Universal Robots PolyScope program: faichun_snake3.urp

Program faichun_snake3 (installation=default directory=/programs/snake_new createdIn=5.11.9.1010452 lastSavedIn=5.11.9.1010452 robotSerialNumber=20225200364)
Calibrated DH parameters: a=[0.00002, -0.569483, -0.54992, -0.00001, -0.000036, 0]; d=[0.180894, -146.691669, 192.918669, -46.053088, 0.119778, 0.115602]; alpha=[1.571425, -0.001534, 0.003359, 1.568739, -1.571477, 0]; deltaTheta=[0, 0.376258, -0.101074, -0.275185, -0.000002, 0]
Robot Program (runOnlyOnce=true)
  Script file /programs/FaiChun_9 Jan_11_2_t1_2.script
    | def Machining1():
    |   # Default parameters:
    |   global speed_ms = 0.05
    |   global speed_rads = 0.75
    |   global accel_mss = 3
    |   global accel_radss = 1.2
    |   global blend_radius_m = 0.0003
    | 
    |   # Add subprograms here
    |   # Start of main program
    |   # Program generated by RoboDK v5.6.8 for UR10e on 17/01/2025 17:23:54
    |   # Using nominal kinematics.
    |   blend_radius_m = 0.0003
    |   speed_ms = 0.05
    |   # set_reference(p[0.340000, -0.238000, 0.001500, 0.000000, 0.000000, 0.000000])
    |   set_tcp(p[0.000000, 0.000000, 0.252000, 0.000000, 0.000000, 0.000000])
    |   # Show Tool
    |   movej([0.145114, -1.397514, -2.446396, -0.868479, 1.570796, 1.715910],accel_radss,speed_rads,0,blend_radius_m)
    |   movel([0.145114, -1.450226, -2.476289, -0.785874, 1.570796, 1.715910],accel_mss,speed_ms,0,blend_radius_m)
    |   #SetTool1
    |   #M_RunCode6
    |   #SetRPM60000
    |   speed_ms = 0.05
    |   #M_RunCode3
    |   movel([0.145114, -1.473196, -2.487384, -0.751808, 1.570796, 1.715910],accel_mss,speed_ms,0,blend_radius_m)
    |   speed_ms = 0.003
    |   movel([0.145114, -1.479129, -2.490086, -0.743174, 1.570796, 1.715910],accel_mss,speed_ms,0,blend_radius_m)
    |   speed_ms = 0.05
    |   movel([-0.131626, -1.561533, -2.414291, -0.736565, 1.570796, 1.439170],accel_mss,speed_ms,0,blend_radius_m)
    |   movel([-0.177704, -1.331249, -2.600139, -0.781001, 1.570796, 1.393092],accel_mss,speed_ms,0,blend_radius_m)
    |   movel([0.204954, -1.166991, -2.688242, -0.857156, 1.570796, 1.775750],accel_mss,speed_ms,0,blend_radius_m)
    |   movel([0.145114, -1.479129, -2.490086, -0.743174, 1.570796, 1.715910],accel_mss,speed_ms,0,blend_radius_m)
    |   speed_ms = 0.003
    |   movel([0.145114, -1.473196, -2.487384, -0.751808, 1.570796, 1.715910],accel_mss,speed_ms,0,blend_radius_m)
    |   speed_ms = 0.05
    |   movel([0.145114, -1.450226, -2.476289, -0.785874, 1.570796, 1.715910],accel_mss,speed_ms,0,blend_radius_m)
    |   #M_RunCode9
    |   movel([0.141001, -1.443521, -2.481739, -0.787129, 1.570796, 1.711798],accel_mss,speed_ms,0,blend_radius_m)
    |   #M_RunCode3
    |   movel([0.141001, -1.466629, -2.492914, -0.752846, 1.570796, 1.711798],accel_mss,speed_ms,0,blend_radius_m)
    |   speed_ms = 0.003
    |   movel([0.141001, -1.472599, -2.495635, -0.744154, 1.570796, 1.711798],accel_mss,speed_ms,0,blend_radius_m)
    |   speed_ms = 0.012
    |   movel([0.136639, -1.473494, -2.494879, -0.744016, 1.570796, 1.707435],accel_mss,speed_ms,0,blend_radius_m)
    |   movel([0.136042, -1.477254, -2.491686, -0.743449, 1.570796, 1.706838],accel_mss,speed_ms,0,blend_radius_m)
    |   movel([0.129615, -1.478592, -2.490545, -0.743252, 1.570796, 1.700411],accel_mss,speed_ms,0,blend_radius_m)
    |   movel([0.130181, -1.474842, -2.493736, -0.743810, 1.570796, 1.700977],accel_mss,speed_ms,0,blend_radius_m)
    |   movel([0.127919, -1.475323, -2.493329, -0.743738, 1.570796, 1.698716],accel_mss,speed_ms,0,blend_radius_m)
    |   movel([0.127361, -1.479068, -2.490138, -0.743183, 1.570796, 1.698157],accel_mss,speed_ms,0,blend_radius_m)
    |   movel([0.121982, -1.480222, -2.489150, -0.743016, 1.570796, 1.692778],accel_mss,speed_ms,0,blend_radius_m)
    |   movel([0.120939, -1.480446, -2.488958, -0.742984, 1.570796, 1.691735],accel_mss,speed_ms,0,blend_radius_m)
    |   movel([0.121724, -1.474915, -2.493675, -0.743799, 1.570796, 1.692520],accel_mss,speed_ms,0,blend_radius_m)
    |   movel([0.126089, -1.473968, -2.494478, -0.743944, 1.570796, 1.696886],accel_mss,speed_ms,0,blend_radius_m)
    |   movel([0.126378, -1.472012, -2.496131, -0.744246, 1.570796, 1.697174],accel_mss,speed_ms,0,blend_radius_m)
    |   movel([0.119733, -1.473463, -2.494905, -0.744021, 1.570796, 1.690529],accel_mss,speed_ms,0,blend_radius_m)
    |   movel([0.118690, -1.480938, -2.488537, -0.742914, 1.570796, 1.689486],accel_mss,speed_ms,0,blend_radius_m)
    |   movel([0.117647, -1.481168, -2.488339, -0.742882, 1.570796, 1.688443],accel_mss,speed_ms,0,blend_radius_m)
    |   speed_ms = 0.02
    |   movel([0.002864, -1.511155, -2.461903, -0.739330, 1.570796, 1.573661],accel_mss,speed_ms,0,blend_radius_m)
    |   movel([-0.108286, -1.549104, -2.426413, -0.736872, 1.570796, 1.462510],accel_mss,speed_ms,0,blend_radius_m)
    |   speed_ms = 0.012
    |   movel([-0.109170, -1.542784, -2.432482, -0.737123, 1.570796, 1.461626],accel_mss,speed_ms,0,blend_radius_m)
    |   movel([-0.115268, -1.545135, -2.430232, -0.737022, 1.570796, 1.455529],accel_mss,speed_ms,0,blend_radius_m)
    |   movel([-0.115029, -1.546770, -2.428662, -0.736957, 1.570796, 1.455767],accel_mss,speed_ms,0,blend_radius_m)
    |   movel([-0.111023, -1.545226, -2.430145, -0.737018, 1.570796, 1.459773],accel_mss,speed_ms,0,blend_radius_m)
    |   movel([-0.110365, -1.549892, -2.425652, -0.736845, 1.570796, 1.460431],accel_mss,speed_ms,0,blend_radius_m)
    |   movel([-0.111325, -1.550258, -2.425297, -0.736833, 1.570796, 1.459472],accel_mss,speed_ms,0,blend_radius_m)
    |   movel([-0.116260, -1.552156, -2.423459, -0.736774, 1.570796, 1.454536],accel_mss,speed_ms,0,blend_radius_m)
    |   movel([-0.116726, -1.549025, -2.426489, -0.736875, 1.570796, 1.454070],accel_mss,speed_ms,0,blend_radius_m)
    |   movel([-0.118795, -1.549827, -2.425715, -0.736847, 1.570796, 1.452001],accel_mss,speed_ms,0,blend_radius_m)
    |   movel([-0.118321, -1.552953, -2.422685, -0.736751, 1.570796, 1.452475],accel_mss,speed_ms,0,blend_radius_m)
    |   movel([-0.124187, -1.555237, -2.420462, -0.736690, 1.570796, 1.446609],accel_mss,speed_ms,0,blend_radius_m)
    |   movel([-0.124683, -1.552129, -2.423485, -0.736775, 1.570796, 1.446114],accel_mss,speed_ms,0,blend_radius_m)
    |   movel([-0.128648, -1.553694, -2.421965, -0.736730, 1.570796, 1.442148],accel_mss,speed_ms,0,blend_radius_m)
    |   movel([-0.129411, -1.549091, -2.426425, -0.736873, 1.570796, 1.441385],accel_mss,speed_ms,0,blend_radius_m)
    |   movel([-0.125425, -1.547510, -2.427949, -0.736929, 1.570796, 1.445371],accel_mss,speed_ms,0,blend_radius_m)
    |   movel([-0.125687, -1.545886, -2.429511, -0.736992, 1.570796, 1.445109],accel_mss,speed_ms,0,blend_radius_m)
    |   movel([-0.129681, -1.547471, -2.427987, -0.736931, 1.570796, 1.441115],accel_mss,speed_ms,0,blend_radius_m)
    |   movel([-0.130331, -1.543596, -2.431706, -0.737087, 1.570796, 1.440465],accel_mss,speed_ms,0,blend_radius_m)
    |   movel([-0.130456, -1.542840, -2.432429, -0.737120, 1.570796, 1.440341],accel_mss,speed_ms,0,blend_radius_m)
    |   movel([-0.124505, -1.540465, -2.434693, -0.737231, 1.570796, 1.446291],accel_mss,speed_ms,0,blend_radius_m)
    |   movel([-0.124003, -1.543613, -2.431690, -0.737086, 1.570796, 1.446793],accel_mss,speed_ms,0,blend_radius_m)
    |   movel([-0.121918, -1.542790, -2.432476, -0.737122, 1.570796, 1.448878],accel_mss,speed_ms,0,blend_radius_m)
    |   movel([-0.122672, -1.537996, -2.437038, -0.737355, 1.570796, 1.448124],accel_mss,speed_ms,0,blend_radius_m)
    |   movel([-0.130730, -1.541209, -2.433985, -0.737195, 1.570796, 1.440067],accel_mss,speed_ms,0,blend_radius_m)
    |   movel([-0.146735, -1.452072, -2.512652, -0.747665, 1.570796, 1.424062],accel_mss,speed_ms,0,blend_radius_m)
    |   speed_ms = 0.02
    |   movel([-0.166789, -1.353893, -2.585329, -0.773167, 1.570796, 1.404008],accel_mss,speed_ms,0,blend_radius_m)
    |   movel([-0.166990, -1.352958, -2.585955, -0.773476, 1.570796, 1.403806],accel_mss,speed_ms,0,blend_radius_m)
    |   speed_ms = 0.012
    |   movel([-0.156896, -1.347760, -2.589410, -0.775219, 1.570796, 1.413900],accel_mss,speed_ms,0,blend_radius_m)
    |   movel([-0.158123, -1.341762, -2.593351, -0.777277, 1.570796, 1.412674],accel_mss,speed_ms,0,blend_radius_m)
    |   movel([-0.160766, -1.343128, -2.592457, -0.776804, 1.570796, 1.410031],accel_mss,speed_ms,0,blend_radius_m)
    |   movel([-0.159947, -1.347068, -2.589867, -0.775454, 1.570796, 1.410849],accel_mss,speed_ms,0,blend_radius_m)
    |   movel([-0.167424, -1.350932, -2.587305, -0.774151, 1.570796, 1.403372],accel_mss,speed_ms,0,blend_radius_m)
    |   movel([-0.167629, -1.349998, -2.587927, -0.774464, 1.570796, 1.403168],accel_mss,speed_ms,0,blend_radius_m)
    |   movel([-0.168693, -1.345153, -2.591129, -0.776107, 1.570796, 1.402103],accel_mss,speed_ms,0,blend_radius_m)
    |   movel([-0.163615, -1.342502, -2.592867, -0.777020, 1.570796, 1.407181],accel_mss,speed_ms,0,blend_radius_m)
    |   movel([-0.164053, -1.340454, -2.594203, -0.777732, 1.570796, 1.406744],accel_mss,speed_ms,0,blend_radius_m)
    |   movel([-0.169143, -1.343118, -2.592464, -0.776807, 1.570796, 1.401654],accel_mss,speed_ms,0,blend_radius_m)
    |   movel([-0.170437, -1.337285, -2.596260, -0.778844, 1.570796, 1.400359],accel_mss,speed_ms,0,blend_radius_m)
    |   movel([-0.165313, -1.334580, -2.598005, -0.779805, 1.570796, 1.405484],accel_mss,speed_ms,0,blend_radius_m)
    |   movel([-0.166173, -1.330591, -2.600559, -0.781239, 1.570796, 1.404623],accel_mss,speed_ms,0,blend_radius_m)
    |   movel([-0.158508, -1.326548, -2.603127, -0.782714, 1.570796, 1.412289],accel_mss,speed_ms,0,blend_radius_m)
    |   movel([-0.157682, -1.330578, -2.600567, -0.781243, 1.570796, 1.413114],accel_mss,speed_ms,0,blend_radius_m)
    |   movel([-0.154998, -1.329179, -2.601459, -0.781752, 1.570796, 1.415798],accel_mss,speed_ms,0,blend_radius_m)
    |   movel([-0.155811, -1.325133, -2.604020, -0.783236, 1.570796, 1.414985],accel_mss,speed_ms,0,blend_radius_m)
    |   movel([-0.148083, -1.321101, -2.606551, -0.784737, 1.570796, 1.422714],accel_mss,speed_ms,0,blend_radius_m)
    |   movel([-0.146935, -1.327148, -2.602747, -0.782494, 1.570796, 1.423861],accel_mss,speed_ms,0,blend_radius_m)
    |   movel([-0.152123, -1.329828, -2.601046, -0.781516, 1.570796, 1.418673],accel_mss,speed_ms,0,blend_radius_m)
    |   movel([-0.151712, -1.331924, -2.599708, -0.780757, 1.570796, 1.419084],accel_mss,speed_ms,0,blend_radius_m)
    |   movel([-0.143841, -1.327877, -2.602285, -0.782227, 1.570796, 1.426955],accel_mss,speed_ms,0,blend_radius_m)
    |   movel([-0.145364, -1.319691, -2.607431, -0.785267, 1.570796, 1.425432],accel_mss,speed_ms,0,blend_radius_m)
    |   movel([0.003920, -1.248574, -2.648506, -0.815310, 1.570796, 1.574716],accel_mss,speed_ms,0,blend_radius_m)
    |   speed_ms = 0.02
    |   movel([0.165154, -1.186625, -2.679348, -0.846417, 1.570796, 1.735951],accel_mss,speed_ms,0,blend_radius_m)
    |   movel([0.163152, -1.198149, -2.673935, -0.840305, 1.570796, 1.733948],accel_mss,speed_ms,0,blend_radius_m)
    |   speed_ms = 0.012
    |   movel([0.172319, -1.195184, -2.675341, -0.841863, 1.570796, 1.743115],accel_mss,speed_ms,0,blend_radius_m)
    |   movel([0.172866, -1.192193, -2.676750, -0.843445, 1.570796, 1.743662],accel_mss,speed_ms,0,blend_radius_m)
    |   movel([0.166811, -1.194153, -2.675828, -0.842408, 1.570796, 1.737608],accel_mss,speed_ms,0,blend_radius_m)
    |   movel([0.168335, -1.185580, -2.679831, -0.846978, 1.570796, 1.739131],accel_mss,speed_ms,0,blend_radius_m)
    |   movel([0.169806, -1.185096, -2.680055, -0.847238, 1.570796, 1.740602],accel_mss,speed_ms,0,blend_radius_m)
    |   movel([0.177391, -1.182622, -2.681194, -0.848573, 1.570796, 1.748187],accel_mss,speed_ms,0,blend_radius_m)
    |   movel([0.176304, -1.188464, -2.678494, -0.845432, 1.570796, 1.747100],accel_mss,speed_ms,0,blend_radius_m)
    |   movel([0.179460, -1.187457, -2.678962, -0.845971, 1.570796, 1.750256],accel_mss,speed_ms,0,blend_radius_m)
    |   movel([0.180574, -1.181595, -2.681665, -0.849129, 1.570796, 1.751371],accel_mss,speed_ms,0,blend_radius_m)
    |   movel([0.189651, -1.178707, -2.682983, -0.850699, 1.570796, 1.760447],accel_mss,speed_ms,0,blend_radius_m)
    |   movel([0.188481, -1.184611, -2.680279, -0.847499, 1.570796, 1.759277],accel_mss,speed_ms,0,blend_radius_m)
    |   movel([0.194577, -1.182720, -2.681149, -0.848520, 1.570796, 1.765374],accel_mss,speed_ms,0,blend_radius_m)
    |   movel([0.192814, -1.191401, -2.677122, -0.843866, 1.570796, 1.763610],accel_mss,speed_ms,0,blend_radius_m)
    |   movel([0.186775, -1.193250, -2.676254, -0.842885, 1.570796, 1.757572],accel_mss,speed_ms,0,blend_radius_m)
    |   movel([0.186185, -1.196251, -2.674837, -0.841302, 1.570796, 1.756982],accel_mss,speed_ms,0,blend_radius_m)
    |   movel([0.192203, -1.194418, -2.675703, -0.842268, 1.570796, 1.762999],accel_mss,speed_ms,0,blend_radius_m)
    |   movel([0.190761, -1.201563, -2.672304, -0.838522, 1.570796, 1.761557],accel_mss,speed_ms,0,blend_radius_m)
    |   movel([0.190484, -1.202941, -2.671643, -0.837806, 1.570796, 1.761280],accel_mss,speed_ms,0,blend_radius_m)
    |   movel([0.181657, -1.205609, -2.670355, -0.836426, 1.570796, 1.752453],accel_mss,speed_ms,0,blend_radius_m)
    |   movel([0.182758, -1.199906, -2.673098, -0.839385, 1.570796, 1.753554],accel_mss,speed_ms,0,blend_radius_m)
    |   movel([0.179644, -1.200868, -2.672637, -0.838884, 1.570796, 1.750441],accel_mss,speed_ms,0,blend_radius_m)
    |   movel([0.178007, -1.209492, -2.668466, -0.834430, 1.570796, 1.748803],accel_mss,speed_ms,0,blend_radius_m)
    |   movel([0.189888, -1.205903, -2.670212, -0.836273, 1.570796, 1.760685],accel_mss,speed_ms,0,blend_radius_m)
    |   speed_ms = 0.02
    |   movel([0.163402, -1.343756, -2.592046, -0.776587, 1.570796, 1.734198],accel_mss,speed_ms,0,blend_radius_m)
    |   movel([0.143535, -1.457310, -2.508372, -0.746708, 1.570796, 1.714331],accel_mss,speed_ms,0,blend_radius_m)
    |   speed_ms = 0.012
    |   movel([0.134639, -1.459191, -2.506824, -0.746374, 1.570796, 1.705436],accel_mss,speed_ms,0,blend_radius_m)
    |   movel([0.133732, -1.465007, -2.502005, -0.745377, 1.570796, 1.704528],accel_mss,speed_ms,0,blend_radius_m)
    |   movel([0.136023, -1.464522, -2.502409, -0.745459, 1.570796, 1.706819],accel_mss,speed_ms,0,blend_radius_m)
    |   movel([0.136629, -1.460695, -2.505582, -0.746111, 1.570796, 1.707425],accel_mss,speed_ms,0,blend_radius_m)
    |   movel([0.143192, -1.459319, -2.506719, -0.746352, 1.570796, 1.713988],accel_mss,speed_ms,0,blend_radius_m)
    |   movel([0.143038, -1.460245, -2.505954, -0.746190, 1.570796, 1.713835],accel_mss,speed_ms,0,blend_radius_m)
    |   movel([0.142251, -1.464999, -2.502011, -0.745379, 1.570796, 1.713048],accel_mss,speed_ms,0,blend_radius_m)
    |   movel([0.137849, -1.465911, -2.501251, -0.745227, 1.570796, 1.708646],accel_mss,speed_ms,0,blend_radius_m)
    |   movel([0.137533, -1.467886, -2.499600, -0.744903, 1.570796, 1.708330],accel_mss,speed_ms,0,blend_radius_m)
    |   movel([0.141927, -1.466979, -2.500359, -0.745051, 1.570796, 1.712723],accel_mss,speed_ms,0,blend_radius_m)
    |   movel([0.141001, -1.472599, -2.495635, -0.744154, 1.570796, 1.711798],accel_mss,speed_ms,0,blend_radius_m)
    |   speed_ms = 0.003
    |   movel([0.141001, -1.466629, -2.492914, -0.752846, 1.570796, 1.711798],accel_mss,speed_ms,0,blend_radius_m)
    |   speed_ms = 0.05
    |   movel([0.141001, -1.443521, -2.481739, -0.787129, 1.570796, 1.711798],accel_mss,speed_ms,0,blend_radius_m)
    |   #M_RunCode9
    |   movel([-0.095971, -1.320143, -2.570643, -0.821603, 1.570796, 1.474826],accel_mss,speed_ms,0,blend_radius_m)
    |   #M_RunCode3
    |   # num 0 inside
    |   movel([-0.095971, -1.345583, -2.583353, -0.783454, 1.570796, 1.474826],accel_mss,speed_ms,0,blend_radius_m)
    |   speed_ms = 0.003
    |   movel([-0.095971, -1.352203, -2.586459, -0.773727, 1.570796, 1.474826],accel_mss,speed_ms,0,blend_radius_m)
    |   speed_ms = 0.015
    |   movel([-0.101060, -1.358991, -2.581897, -0.771501, 1.570796, 1.469736],accel_mss,speed_ms,0,blend_radius_m)
    |   movel([-0.105019, -1.363609, -2.578758, -0.770023, 1.570796, 1.465778],accel_mss,speed_ms,0,blend_radius_m)
    |   movel([-0.106639, -1.365123, -2.577722, -0.769544, 1.570796, 1.464157],accel_mss,speed_ms,0,blend_radius_m)
    |   movel([-0.108096, -1.366111, -2.577044, -0.769234, 1.570796, 1.462701],accel_mss,speed_ms,0,blend_radius_m)
    |   movel([-0.109388, -1.366578, -2.576723, -0.769088, 1.570796, 1.461409],accel_mss,speed_ms,0,blend_radius_m)
    |   movel([-0.110520, -1.366524, -2.576760, -0.769105, 1.570796, 1.460276],accel_mss,speed_ms,0,blend_radius_m)
    |   movel([-0.111321, -1.366002, -2.577119, -0.769268, 1.570796, 1.459475],accel_mss,speed_ms,0,blend_radius_m)
    |   movel([-0.111616, -1.365061, -2.577764, -0.769564, 1.570796, 1.459180],accel_mss,speed_ms,0,blend_radius_m)
    |   movel([-0.111403, -1.363700, -2.578696, -0.769994, 1.570796, 1.459393],accel_mss,speed_ms,0,blend_radius_m)
    |   movel([-0.110683, -1.361913, -2.579914, -0.770562, 1.570796, 1.460113],accel_mss,speed_ms,0,blend_radius_m)
    |   movel([-0.107823, -1.356944, -2.583280, -0.772165, 1.570796, 1.462973],accel_mss,speed_ms,0,blend_radius_m)
    |   movel([-0.103126, -1.350010, -2.587919, -0.774460, 1.570796, 1.467671],accel_mss,speed_ms,0,blend_radius_m)
    |   movel([-0.097993, -1.343109, -2.592470, -0.776810, 1.570796, 1.472803],accel_mss,speed_ms,0,blend_radius_m)
    |   movel([-0.093909, -1.338331, -2.595583, -0.778476, 1.570796, 1.476888],accel_mss,speed_ms,0,blend_radius_m)
    |   movel([-0.092221, -1.336752, -2.596604, -0.779033, 1.570796, 1.478576],accel_mss,speed_ms,0,blend_radius_m)
    |   movel([-0.090706, -1.335718, -2.597272, -0.779399, 1.570796, 1.480090],accel_mss,speed_ms,0,blend_radius_m)
    |   movel([-0.089366, -1.335233, -2.597584, -0.779572, 1.570796, 1.481430],accel_mss,speed_ms,0,blend_radius_m)
    |   movel([-0.088203, -1.335298, -2.597543, -0.779549, 1.570796, 1.482593],accel_mss,speed_ms,0,blend_radius_m)
    |   movel([-0.087396, -1.335857, -2.597182, -0.779350, 1.570796, 1.483400],accel_mss,speed_ms,0,blend_radius_m)
    |   movel([-0.087120, -1.336850, -2.596541, -0.778998, 1.570796, 1.483676],accel_mss,speed_ms,0,blend_radius_m)
    |   movel([-0.087378, -1.338279, -2.595616, -0.778494, 1.570796, 1.483418],accel_mss,speed_ms,0,blend_radius_m)
    |   movel([-0.088162, -1.340134, -2.594412, -0.777843, 1.570796, 1.482634],accel_mss,speed_ms,0,blend_radius_m)
    |   movel([-0.091172, -1.345231, -2.591077, -0.776081, 1.570796, 1.479624],accel_mss,speed_ms,0,blend_radius_m)
    |   movel([-0.095971, -1.352203, -2.586459, -0.773727, 1.570796, 1.474826],accel_mss,speed_ms,0,blend_radius_m)
    |   speed_ms = 0.003
    |   movel([-0.095971, -1.345583, -2.583353, -0.783454, 1.570796, 1.474826],accel_mss,speed_ms,0,blend_radius_m)
    |   speed_ms = 0.05
    |   movel([-0.095971, -1.320143, -2.570643, -0.821603, 1.570796, 1.474826],accel_mss,speed_ms,0,blend_radius_m)
    |   #M_RunCode9
    |   movel([-0.088305, -1.322635, -2.569052, -0.820702, 1.570796, 1.482491],accel_mss,speed_ms,0,blend_radius_m)
    |   #M_RunCode3
    |   #num 0 outside
    |   movel([-0.088305, -1.348033, -2.581729, -0.782626, 1.570796, 1.482491],accel_mss,speed_ms,0,blend_radius_m)
    |   speed_ms = 0.003
    |   movel([-0.088305, -1.354642, -2.584827, -0.772920, 1.570796, 1.482491],accel_mss,speed_ms,0,blend_radius_m)
    |   speed_ms = 0.015
    |   movel([-0.090204, -1.357095, -2.583178, -0.772116, 1.570796, 1.480592],accel_mss,speed_ms,0,blend_radius_m)
    |   movel([-0.092146, -1.359299, -2.581689, -0.771401, 1.570796, 1.478650],accel_mss,speed_ms,0,blend_radius_m)
    |   movel([-0.094134, -1.361259, -2.580359, -0.770771, 1.570796, 1.476662],accel_mss,speed_ms,0,blend_radius_m)
    |   movel([-0.096168, -1.362974, -2.579191, -0.770224, 1.570796, 1.474629],accel_mss,speed_ms,0,blend_radius_m)
    |   movel([-0.098207, -1.364435, -2.578193, -0.769761, 1.570796, 1.472589],accel_mss,speed_ms,0,blend_radius_m)
    |   movel([-0.100213, -1.365632, -2.577372, -0.769384, 1.570796, 1.470584],accel_mss,speed_ms,0,blend_radius_m)
    |   movel([-0.102186, -1.366569, -2.576729, -0.769091, 1.570796, 1.468610],accel_mss,speed_ms,0,blend_radius_m)
    |   movel([-0.104128, -1.367242, -2.576266, -0.768881, 1.570796, 1.466669],accel_mss,speed_ms,0,blend_radius_m)
    |   movel([-0.106011, -1.367658, -2.575980, -0.768751, 1.570796, 1.464785],accel_mss,speed_ms,0,blend_radius_m)
    |   movel([-0.107803, -1.367820, -2.575868, -0.768701, 1.570796, 1.462993],accel_mss,speed_ms,0,blend_radius_m)
    |   movel([-0.109510, -1.367730, -2.575930, -0.768729, 1.570796, 1.461286],accel_mss,speed_ms,0,blend_radius_m)
    |   movel([-0.111131, -1.367388, -2.576166, -0.768835, 1.570796, 1.459665],accel_mss,speed_ms,0,blend_radius_m)
    |   movel([-0.112591, -1.366814, -2.576561, -0.769014, 1.570796, 1.458205],accel_mss,speed_ms,0,blend_radius_m)
    |   movel([-0.113810, -1.366033, -2.577098, -0.769259, 1.570796, 1.456987],accel_mss,speed_ms,0,blend_radius_m)
    |   movel([-0.114791, -1.365044, -2.577776, -0.769569, 1.570796, 1.456006],accel_mss,speed_ms,0,blend_radius_m)
    |   movel([-0.115530, -1.363841, -2.578599, -0.769949, 1.570796, 1.455266],accel_mss,speed_ms,0,blend_radius_m)
    |   movel([-0.116005, -1.362439, -2.579556, -0.770394, 1.570796, 1.454792],accel_mss,speed_ms,0,blend_radius_m)
    |   movel([-0.116190, -1.360849, -2.580638, -0.770902, 1.570796, 1.454606],accel_mss,speed_ms,0,blend_radius_m)
    |   movel([-0.116085, -1.359067, -2.581846, -0.771476, 1.570796, 1.454711],accel_mss,speed_ms,0,blend_radius_m)
    |   movel([-0.115685, -1.357091, -2.583180, -0.772117, 1.570796, 1.455111],accel_mss,speed_ms,0,blend_radius_m)
    |   movel([-0.114980, -1.354950, -2.584621, -0.772819, 1.570796, 1.455816],accel_mss,speed_ms,0,blend_radius_m)
    |   movel([-0.113953, -1.352671, -2.586146, -0.773572, 1.570796, 1.456843],accel_mss,speed_ms,0,blend_radius_m)
    |   movel([-0.112603, -1.350256, -2.587755, -0.774378, 1.570796, 1.458193],accel_mss,speed_ms,0,blend_radius_m)
    |   movel([-0.110928, -1.347704, -2.589447, -0.775238, 1.570796, 1.459868],accel_mss,speed_ms,0,blend_radius_m)
    |   movel([-0.109051, -1.345192, -2.591103, -0.776094, 1.570796, 1.461745],accel_mss,speed_ms,0,blend_radius_m)
    |   movel([-0.107107, -1.342916, -2.592596, -0.776877, 1.570796, 1.463689],accel_mss,speed_ms,0,blend_radius_m)
    |   movel([-0.105094, -1.340873, -2.593931, -0.777586, 1.570796, 1.465702],accel_mss,speed_ms,0,blend_radius_m)
    |   movel([-0.103017, -1.339070, -2.595103, -0.778216, 1.570796, 1.467780],accel_mss,speed_ms,0,blend_radius_m)
    |   movel([-0.100919, -1.337525, -2.596105, -0.778759, 1.570796, 1.469878],accel_mss,speed_ms,0,blend_radius_m)
    |   movel([-0.098849, -1.336258, -2.596923, -0.779208, 1.570796, 1.471947],accel_mss,speed_ms,0,blend_radius_m)
    |   movel([-0.096809, -1.335267, -2.597562, -0.779560, 1.570796, 1.473987],accel_mss,speed_ms,0,blend_radius_m)
    |   movel([-0.094800, -1.334558, -2.598018, -0.779812, 1.570796, 1.475997],accel_mss,speed_ms,0,blend_radius_m)
    |   movel([-0.092856, -1.334126, -2.598296, -0.779966, 1.570796, 1.477940],accel_mss,speed_ms,0,blend_radius_m)
    |   movel([-0.091005, -1.333963, -2.598401, -0.780025, 1.570796, 1.479791],accel_mss,speed_ms,0,blend_radius_m)
    |   movel([-0.089247, -1.334068, -2.598334, -0.779987, 1.570796, 1.481550],accel_mss,speed_ms,0,blend_radius_m)
    |   movel([-0.087589, -1.334445, -2.598091, -0.779853, 1.570796, 1.483208],accel_mss,speed_ms,0,blend_radius_m)
    |   movel([-0.086106, -1.335067, -2.597691, -0.779631, 1.570796, 1.484690],accel_mss,speed_ms,0,blend_radius_m)
    |   movel([-0.084880, -1.335904, -2.597152, -0.779333, 1.570796, 1.485916],accel_mss,speed_ms,0,blend_radius_m)
    |   movel([-0.083910, -1.336959, -2.596471, -0.778959, 1.570796, 1.486886],accel_mss,speed_ms,0,blend_radius_m)
    |   movel([-0.083195, -1.338228, -2.595649, -0.778512, 1.570796, 1.487601],accel_mss,speed_ms,0,blend_radius_m)
    |   movel([-0.082761, -1.339697, -2.594696, -0.777996, 1.570796, 1.488035],accel_mss,speed_ms,0,blend_radius_m)
    |   movel([-0.082632, -1.341356, -2.593615, -0.777417, 1.570796, 1.488165],accel_mss,speed_ms,0,blend_radius_m)
    |   movel([-0.082808, -1.343205, -2.592407, -0.776777, 1.570796, 1.487989],accel_mss,speed_ms,0,blend_radius_m)
    |   movel([-0.083285, -1.345236, -2.591074, -0.776079, 1.570796, 1.487512],accel_mss,speed_ms,0,blend_radius_m)
    |   movel([-0.084070, -1.347416, -2.589637, -0.775336, 1.570796, 1.486727],accel_mss,speed_ms,0,blend_radius_m)
    |   movel([-0.085171, -1.349713, -2.588116, -0.774560, 1.570796, 1.485626],accel_mss,speed_ms,0,blend_radius_m)
    |   movel([-0.086583, -1.352122, -2.586513, -0.773754, 1.570796, 1.484213],accel_mss,speed_ms,0,blend_radius_m)
    |   movel([-0.088305, -1.354642, -2.584827, -0.772920, 1.570796, 1.482491],accel_mss,speed_ms,0,blend_radius_m)
    |   speed_ms = 0.003
    |   movel([-0.088305, -1.348033, -2.581729, -0.782626, 1.570796, 1.482491],accel_mss,speed_ms,0,blend_radius_m)
    |   speed_ms = 0.05
    |   movel([-0.088305, -1.322635, -2.569052, -0.820702, 1.570796, 1.482491],accel_mss,speed_ms,0,blend_radius_m)
    |   #M_RunCode9
    |   movel([-0.118832, -1.321958, -2.569485, -0.820946, 1.570796, 1.451964],accel_mss,speed_ms,0,blend_radius_m)
    |   #M_RunCode3
    |   movel([-0.118832, -1.347368, -2.582171, -0.782850, 1.570796, 1.451964],accel_mss,speed_ms,0,blend_radius_m)
    |   speed_ms = 0.003
    |   movel([-0.118832, -1.353979, -2.585271, -0.773138, 1.570796, 1.451964],accel_mss,speed_ms,0,blend_radius_m)
    |   speed_ms = 0.02
    |   movel([-0.124934, -1.362775, -2.579327, -0.770287, 1.570796, 1.445862],accel_mss,speed_ms,0,blend_radius_m)
    |   movel([-0.148632, -1.356620, -2.583498, -0.772271, 1.570796, 1.422164],accel_mss,speed_ms,0,blend_radius_m)
    |   movel([-0.148043, -1.355734, -2.584094, -0.772561, 1.570796, 1.422754],accel_mss,speed_ms,0,blend_radius_m)
    |   movel([-0.146262, -1.353538, -2.585567, -0.773284, 1.570796, 1.424534],accel_mss,speed_ms,0,blend_radius_m)
    |   movel([-0.143953, -1.351516, -2.586917, -0.773956, 1.570796, 1.426844],accel_mss,speed_ms,0,blend_radius_m)
    |   movel([-0.141315, -1.349690, -2.588131, -0.774568, 1.570796, 1.429481],accel_mss,speed_ms,0,blend_radius_m)
    |   movel([-0.138559, -1.348086, -2.589194, -0.775109, 1.570796, 1.432238],accel_mss,speed_ms,0,blend_radius_m)
    |   movel([-0.130967, -1.344319, -2.591676, -0.776393, 1.570796, 1.439829],accel_mss,speed_ms,0,blend_radius_m)
    |   movel([-0.123880, -1.340890, -2.593919, -0.777580, 1.570796, 1.446916],accel_mss,speed_ms,0,blend_radius_m)
    |   movel([-0.121261, -1.339412, -2.594881, -0.778096, 1.570796, 1.449535],accel_mss,speed_ms,0,blend_radius_m)
    |   movel([-0.118795, -1.337754, -2.595956, -0.778678, 1.570796, 1.452001],accel_mss,speed_ms,0,blend_radius_m)
    |   movel([-0.116656, -1.335945, -2.597125, -0.779319, 1.570796, 1.454140],accel_mss,speed_ms,0,blend_radius_m)
    |   movel([-0.115017, -1.334007, -2.598373, -0.780009, 1.570796, 1.455779],accel_mss,speed_ms,0,blend_radius_m)
    |   movel([-0.113700, -1.331542, -2.599952, -0.780895, 1.570796, 1.457096],accel_mss,speed_ms,0,blend_radius_m)
    |   movel([-0.113452, -1.330481, -2.600629, -0.781279, 1.570796, 1.457345],accel_mss,speed_ms,0,blend_radius_m)
    |   movel([-0.113477, -1.329535, -2.601232, -0.781622, 1.570796, 1.457320],accel_mss,speed_ms,0,blend_radius_m)
    |   movel([-0.114162, -1.328078, -2.602158, -0.782154, 1.570796, 1.456635],accel_mss,speed_ms,0,blend_radius_m)
    |   movel([-0.115566, -1.327268, -2.602671, -0.782450, 1.570796, 1.455230],accel_mss,speed_ms,0,blend_radius_m)
    |   movel([-0.116775, -1.327100, -2.602777, -0.782511, 1.570796, 1.454022],accel_mss,speed_ms,0,blend_radius_m)
    |   movel([-0.117884, -1.327287, -2.602659, -0.782443, 1.570796, 1.452913],accel_mss,speed_ms,0,blend_radius_m)
    |   movel([-0.118818, -1.327765, -2.602356, -0.782268, 1.570796, 1.451978],accel_mss,speed_ms,0,blend_radius_m)
    |   movel([-0.119500, -1.328465, -2.601912, -0.782012, 1.570796, 1.451297],accel_mss,speed_ms,0,blend_radius_m)
    |   movel([-0.119848, -1.329672, -2.601145, -0.781572, 1.570796, 1.450949],accel_mss,speed_ms,0,blend_radius_m)
    |   movel([-0.120081, -1.330839, -2.600401, -0.781149, 1.570796, 1.450715],accel_mss,speed_ms,0,blend_radius_m)
    |   movel([-0.120851, -1.332269, -2.599487, -0.780633, 1.570796, 1.449945],accel_mss,speed_ms,0,blend_radius_m)
    |   movel([-0.122252, -1.333823, -2.598491, -0.780075, 1.570796, 1.448544],accel_mss,speed_ms,0,blend_radius_m)
    |   movel([-0.123926, -1.334807, -2.597858, -0.779723, 1.570796, 1.446870],accel_mss,speed_ms,0,blend_radius_m)
    |   movel([-0.125677, -1.335229, -2.597587, -0.779573, 1.570796, 1.445119],accel_mss,speed_ms,0,blend_radius_m)
    |   movel([-0.127302, -1.335096, -2.597672, -0.779620, 1.570796, 1.443494],accel_mss,speed_ms,0,blend_radius_m)
    |   movel([-0.128587, -1.334465, -2.598078, -0.779846, 1.570796, 1.442210],accel_mss,speed_ms,0,blend_radius_m)
    |   movel([-0.129320, -1.333388, -2.598770, -0.780231, 1.570796, 1.441477],accel_mss,speed_ms,0,blend_radius_m)
    |   movel([-0.129352, -1.331950, -2.599691, -0.780748, 1.570796, 1.441444],accel_mss,speed_ms,0,blend_radius_m)
    |   movel([-0.128528, -1.330238, -2.600784, -0.781367, 1.570796, 1.442268],accel_mss,speed_ms,0,blend_radius_m)
    |   movel([-0.127385, -1.328836, -2.601677, -0.781877, 1.570796, 1.443412],accel_mss,speed_ms,0,blend_radius_m)
    |   movel([-0.126030, -1.327695, -2.602400, -0.782293, 1.570796, 1.444766],accel_mss,speed_ms,0,blend_radius_m)
    |   movel([-0.124463, -1.326815, -2.602958, -0.782616, 1.570796, 1.446334],accel_mss,speed_ms,0,blend_radius_m)
    |   movel([-0.122683, -1.326203, -2.603345, -0.782841, 1.570796, 1.448113],accel_mss,speed_ms,0,blend_radius_m)
    |   movel([-0.120785, -1.325853, -2.603565, -0.782970, 1.570796, 1.450011],accel_mss,speed_ms,0,blend_radius_m)
    |   movel([-0.118858, -1.325758, -2.603626, -0.783005, 1.570796, 1.451938],accel_mss,speed_ms,0,blend_radius_m)
    |   movel([-0.114926, -1.326342, -2.603257, -0.782790, 1.570796, 1.455870],accel_mss,speed_ms,0,blend_radius_m)
    |   movel([-0.112673, -1.327135, -2.602755, -0.782499, 1.570796, 1.458123],accel_mss,speed_ms,0,blend_radius_m)
    |   movel([-0.110749, -1.328180, -2.602093, -0.782116, 1.570796, 1.460048],accel_mss,speed_ms,0,blend_radius_m)
    |   movel([-0.109155, -1.329474, -2.601271, -0.781644, 1.570796, 1.461641],accel_mss,speed_ms,0,blend_radius_m)
    |   movel([-0.107892, -1.331014, -2.600289, -0.781086, 1.570796, 1.462904],accel_mss,speed_ms,0,blend_radius_m)
    |   movel([-0.107162, -1.332798, -2.599148, -0.780443, 1.570796, 1.463634],accel_mss,speed_ms,0,blend_radius_m)
    |   movel([-0.107176, -1.334831, -2.597843, -0.779715, 1.570796, 1.463620],accel_mss,speed_ms,0,blend_radius_m)
    |   movel([-0.107927, -1.337107, -2.596375, -0.778907, 1.570796, 1.462869],accel_mss,speed_ms,0,blend_radius_m)
    |   movel([-0.109406, -1.339620, -2.594746, -0.778023, 1.570796, 1.461391],accel_mss,speed_ms,0,blend_radius_m)
    |   movel([-0.111183, -1.341801, -2.593325, -0.777263, 1.570796, 1.459613],accel_mss,speed_ms,0,blend_radius_m)
    |   movel([-0.113261, -1.343698, -2.592084, -0.776607, 1.570796, 1.457535],accel_mss,speed_ms,0,blend_radius_m)
    |   movel([-0.115524, -1.345335, -2.591009, -0.776045, 1.570796, 1.455272],accel_mss,speed_ms,0,blend_radius_m)
    |   movel([-0.117852, -1.346735, -2.590087, -0.775567, 1.570796, 1.452944],accel_mss,speed_ms,0,blend_radius_m)
    |   movel([-0.123738, -1.349638, -2.588166, -0.774585, 1.570796, 1.447059],accel_mss,speed_ms,0,blend_radius_m)
    |   movel([-0.129266, -1.352407, -2.586322, -0.773659, 1.570796, 1.441530],accel_mss,speed_ms,0,blend_radius_m)
    |   movel([-0.131364, -1.353673, -2.585476, -0.773239, 1.570796, 1.439432],accel_mss,speed_ms,0,blend_radius_m)
    |   movel([-0.133365, -1.355125, -2.584503, -0.772761, 1.570796, 1.437431],accel_mss,speed_ms,0,blend_radius_m)
    |   movel([-0.135159, -1.356768, -2.583398, -0.772223, 1.570796, 1.435638],accel_mss,speed_ms,0,blend_radius_m)
    |   movel([-0.136628, -1.358602, -2.582161, -0.771626, 1.570796, 1.434168],accel_mss,speed_ms,0,blend_radius_m)
    |   movel([-0.135740, -1.358833, -2.582004, -0.771552, 1.570796, 1.435057],accel_mss,speed_ms,0,blend_radius_m)
    |   movel([-0.133192, -1.359344, -2.581658, -0.771387, 1.570796, 1.437605],accel_mss,speed_ms,0,blend_radius_m)
    |   movel([-0.130761, -1.359508, -2.581548, -0.771334, 1.570796, 1.440035],accel_mss,speed_ms,0,blend_radius_m)
    |   movel([-0.128449, -1.359327, -2.581670, -0.771392, 1.570796, 1.442347],accel_mss,speed_ms,0,blend_radius_m)
    |   movel([-0.126248, -1.358795, -2.582030, -0.771564, 1.570796, 1.444548],accel_mss,speed_ms,0,blend_radius_m)
    |   movel([-0.124179, -1.357967, -2.582590, -0.771832, 1.570796, 1.446617],accel_mss,speed_ms,0,blend_radius_m)
    |   movel([-0.122254, -1.356890, -2.583316, -0.772183, 1.570796, 1.448542],accel_mss,speed_ms,0,blend_radius_m)
    |   movel([-0.120474, -1.355562, -2.584210, -0.772617, 1.570796, 1.450322],accel_mss,speed_ms,0,blend_radius_m)
    |   movel([-0.118832, -1.353979, -2.585271, -0.773138, 1.570796, 1.451964],accel_mss,speed_ms,0,blend_radius_m)
    |   speed_ms = 0.003
    |   movel([-0.118832, -1.347368, -2.582171, -0.782850, 1.570796, 1.451964],accel_mss,speed_ms,0,blend_radius_m)
    |   speed_ms = 0.05
    |   movel([-0.118832, -1.321958, -2.569485, -0.820946, 1.570796, 1.451964],accel_mss,speed_ms,0,blend_radius_m)
    |   #M_RunCode9
    |   movel([0.073358, -1.418214, -2.501717, -0.792458, 1.570796, 1.644154],accel_mss,speed_ms,0,blend_radius_m)
    |   #M_RunCode3
    |   movel([0.073358, -1.441837, -2.513195, -0.757357, 1.570796, 1.644154],accel_mss,speed_ms,0,blend_radius_m)
    |   speed_ms = 0.003
    |   movel([0.073358, -1.447948, -2.515992, -0.748448, 1.570796, 1.644154],accel_mss,speed_ms,0,blend_radius_m)
    |   speed_ms = 0.02
    |   movel([0.075270, -1.446294, -2.517325, -0.748770, 1.570796, 1.646066],accel_mss,speed_ms,0,blend_radius_m)
    |   movel([0.077554, -1.444921, -2.518428, -0.749040, 1.570796, 1.648350],accel_mss,speed_ms,0,blend_radius_m)
    |   movel([0.080047, -1.443807, -2.519321, -0.749261, 1.570796, 1.650843],accel_mss,speed_ms,0,blend_radius_m)
    |   movel([0.082577, -1.442932, -2.520021, -0.749436, 1.570796, 1.653374],accel_mss,speed_ms,0,blend_radius_m)
    |   movel([0.089381, -1.441132, -2.521457, -0.749800, 1.570796, 1.660178],accel_mss,speed_ms,0,blend_radius_m)
    |   movel([0.095696, -1.439540, -2.522724, -0.750126, 1.570796, 1.666492],accel_mss,speed_ms,0,blend_radius_m)
    |   movel([0.098074, -1.438760, -2.523343, -0.750287, 1.570796, 1.668870],accel_mss,speed_ms,0,blend_radius_m)
    |   movel([0.100372, -1.437779, -2.524119, -0.750490, 1.570796, 1.671168],accel_mss,speed_ms,0,blend_radius_m)
    |   movel([0.102449, -1.436586, -2.525063, -0.750740, 1.570796, 1.673245],accel_mss,speed_ms,0,blend_radius_m)
    |   movel([0.104165, -1.435162, -2.526185, -0.751041, 1.570796, 1.674961],accel_mss,speed_ms,0,blend_radius_m)
    |   movel([0.105751, -1.433181, -2.527743, -0.751465, 1.570796, 1.676547],accel_mss,speed_ms,0,blend_radius_m)
    |   movel([0.106187, -1.432257, -2.528467, -0.751665, 1.570796, 1.676983],accel_mss,speed_ms,0,blend_radius_m)
    |   movel([0.106384, -1.431377, -2.529156, -0.751856, 1.570796, 1.677181],accel_mss,speed_ms,0,blend_radius_m)
    |   movel([0.106189, -1.429873, -2.530330, -0.752186, 1.570796, 1.676986],accel_mss,speed_ms,0,blend_radius_m)
    |   movel([0.105289, -1.428805, -2.531162, -0.752422, 1.570796, 1.676086],accel_mss,speed_ms,0,blend_radius_m)
    |   movel([0.104393, -1.428371, -2.531499, -0.752519, 1.570796, 1.675190],accel_mss,speed_ms,0,blend_radius_m)
    |   movel([0.103490, -1.428293, -2.531560, -0.752536, 1.570796, 1.674286],accel_mss,speed_ms,0,blend_radius_m)
    |   movel([0.102658, -1.428519, -2.531384, -0.752486, 1.570796, 1.673455],accel_mss,speed_ms,0,blend_radius_m)
    |   movel([0.101969, -1.429012, -2.531001, -0.752376, 1.570796, 1.672765],accel_mss,speed_ms,0,blend_radius_m)
    |   movel([0.101420, -1.430050, -2.530192, -0.752147, 1.570796, 1.672216],accel_mss,speed_ms,0,blend_radius_m)
    |   movel([0.100969, -1.431080, -2.529388, -0.751921, 1.570796, 1.671765],accel_mss,speed_ms,0,blend_radius_m)
    |   movel([0.100039, -1.432229, -2.528489, -0.751671, 1.570796, 1.670835],accel_mss,speed_ms,0,blend_radius_m)
    |   movel([0.098595, -1.433352, -2.527609, -0.751428, 1.570796, 1.669391],accel_mss,speed_ms,0,blend_radius_m)
    |   movel([0.097067, -1.433883, -2.527192, -0.751314, 1.570796, 1.667864],accel_mss,speed_ms,0,blend_radius_m)
    |   movel([0.095608, -1.433877, -2.527196, -0.751315, 1.570796, 1.666404],accel_mss,speed_ms,0,blend_radius_m)
    |   movel([0.094378, -1.433385, -2.527583, -0.751421, 1.570796, 1.665174],accel_mss,speed_ms,0,blend_radius_m)
    |   movel([0.093528, -1.432503, -2.528274, -0.751611, 1.570796, 1.664324],accel_mss,speed_ms,0,blend_radius_m)
    |   movel([0.093210, -1.431334, -2.529189, -0.751866, 1.570796, 1.664006],accel_mss,speed_ms,0,blend_radius_m)
    |   movel([0.093521, -1.429992, -2.530237, -0.752160, 1.570796, 1.664317],accel_mss,speed_ms,0,blend_radius_m)
    |   movel([0.094560, -1.428589, -2.531329, -0.752470, 1.570796, 1.665357],accel_mss,speed_ms,0,blend_radius_m)
    |   movel([0.095773, -1.427547, -2.532139, -0.752703, 1.570796, 1.666569],accel_mss,speed_ms,0,blend_radius_m)
    |   movel([0.097091, -1.426799, -2.532719, -0.752871, 1.570796, 1.667888],accel_mss,speed_ms,0,blend_radius_m)
    |   movel([0.098510, -1.426345, -2.533071, -0.752973, 1.570796, 1.669306],accel_mss,speed_ms,0,blend_radius_m)
    |   movel([0.100028, -1.426187, -2.533193, -0.753009, 1.570796, 1.670824],accel_mss,speed_ms,0,blend_radius_m)
    |   movel([0.101578, -1.426298, -2.533108, -0.752984, 1.570796, 1.672374],accel_mss,speed_ms,0,blend_radius_m)
    |   movel([0.103090, -1.426654, -2.532832, -0.752903, 1.570796, 1.673886],accel_mss,speed_ms,0,blend_radius_m)
    |   movel([0.105998, -1.428092, -2.531716, -0.752581, 1.570796, 1.676795],accel_mss,speed_ms,0,blend_radius_m)
    |   movel([0.107557, -1.429342, -2.530744, -0.752303, 1.570796, 1.678354],accel_mss,speed_ms,0,blend_radius_m)
    |   movel([0.108806, -1.430745, -2.529650, -0.751994, 1.570796, 1.679602],accel_mss,speed_ms,0,blend_radius_m)
    |   movel([0.109743, -1.432300, -2.528433, -0.751655, 1.570796, 1.680539],accel_mss,speed_ms,0,blend_radius_m)
    |   movel([0.110369, -1.434007, -2.527094, -0.751288, 1.570796, 1.681165],accel_mss,speed_ms,0,blend_radius_m)
    |   movel([0.110526, -1.435818, -2.525669, -0.750902, 1.570796, 1.681322],accel_mss,speed_ms,0,blend_radius_m)
    |   movel([0.110053, -1.437690, -2.524190, -0.750509, 1.570796, 1.680850],accel_mss,speed_ms,0,blend_radius_m)
    |   movel([0.108957, -1.439621, -2.522659, -0.750109, 1.570796, 1.679754],accel_mss,speed_ms,0,blend_radius_m)
    |   movel([0.107237, -1.441611, -2.521075, -0.749702, 1.570796, 1.678034],accel_mss,speed_ms,0,blend_radius_m)
    |   movel([0.105364, -1.443229, -2.519783, -0.749376, 1.570796, 1.676160],accel_mss,speed_ms,0,blend_radius_m)
    |   movel([0.103317, -1.444521, -2.518749, -0.749119, 1.570796, 1.674113],accel_mss,speed_ms,0,blend_radius_m)
    |   movel([0.101180, -1.445533, -2.517936, -0.748919, 1.570796, 1.671977],accel_mss,speed_ms,0,blend_radius_m)
    |   movel([0.099050, -1.446312, -2.517311, -0.748766, 1.570796, 1.669846],accel_mss,speed_ms,0,blend_radius_m)
    |   movel([0.093795, -1.447697, -2.516195, -0.748497, 1.570796, 1.664592],accel_mss,speed_ms,0,blend_radius_m)
    |   movel([0.088839, -1.449042, -2.515109, -0.748238, 1.570796, 1.659636],accel_mss,speed_ms,0,blend_radius_m)
    |   movel([0.086906, -1.449752, -2.514535, -0.748103, 1.570796, 1.657703],accel_mss,speed_ms,0,blend_radius_m)
    |   movel([0.085004, -1.450661, -2.513798, -0.747930, 1.570796, 1.655801],accel_mss,speed_ms,0,blend_radius_m)
    |   movel([0.083219, -1.451795, -2.512877, -0.747717, 1.570796, 1.654015],accel_mss,speed_ms,0,blend_radius_m)
    |   movel([0.081643, -1.453180, -2.511750, -0.747459, 1.570796, 1.652439],accel_mss,speed_ms,0,blend_radius_m)
    |   movel([0.082284, -1.453594, -2.511413, -0.747383, 1.570796, 1.653080],accel_mss,speed_ms,0,blend_radius_m)
    |   movel([0.084167, -1.454631, -2.510566, -0.747192, 1.570796, 1.654964],accel_mss,speed_ms,0,blend_radius_m)
    |   movel([0.086036, -1.455322, -2.510001, -0.747066, 1.570796, 1.656832],accel_mss,speed_ms,0,blend_radius_m)
    |   movel([0.087890, -1.455663, -2.509722, -0.747004, 1.570796, 1.658686],accel_mss,speed_ms,0,blend_radius_m)
    |   movel([0.089734, -1.455653, -2.509730, -0.747006, 1.570796, 1.660530],accel_mss,speed_ms,0,blend_radius_m)
    |   movel([0.091546, -1.455337, -2.509989, -0.747063, 1.570796, 1.662343],accel_mss,speed_ms,0,blend_radius_m)
    |   movel([0.093297, -1.454760, -2.510461, -0.747169, 1.570796, 1.664093],accel_mss,speed_ms,0,blend_radius_m)
    |   movel([0.094994, -1.453918, -2.511148, -0.747323, 1.570796, 1.665790],accel_mss,speed_ms,0,blend_radius_m)
    |   movel([0.096635, -1.452811, -2.512050, -0.747527, 1.570796, 1.667431],accel_mss,speed_ms,0,blend_radius_m)
    |   movel([0.089860, -1.459642, -2.506452, -0.746295, 1.570796, 1.660656],accel_mss,speed_ms,0,blend_radius_m)
    |   movel([0.072686, -1.448648, -2.515427, -0.748314, 1.570796, 1.643483],accel_mss,speed_ms,0,blend_radius_m)
    |   movel([0.073358, -1.447948, -2.515992, -0.748448, 1.570796, 1.644154],accel_mss,speed_ms,0,blend_radius_m)
    |   speed_ms = 0.003
    |   movel([0.073358, -1.441837, -2.513195, -0.757357, 1.570796, 1.644154],accel_mss,speed_ms,0,blend_radius_m)
    |   speed_ms = 0.05
    |   movel([0.073358, -1.418214, -2.501717, -0.792458, 1.570796, 1.644154],accel_mss,speed_ms,0,blend_radius_m)
    |   #M_RunCode9
    |   movel([0.096184, -1.427284, -2.494664, -0.790441, 1.570796, 1.666981],accel_mss,speed_ms,0,blend_radius_m)
    |   #M_RunCode3
    |   movel([0.096184, -1.450724, -2.506032, -0.755633, 1.570796, 1.666981],accel_mss,speed_ms,0,blend_radius_m)
    |   speed_ms = 0.003
    |   movel([0.096184, -1.456785, -2.508802, -0.746802, 1.570796, 1.666981],accel_mss,speed_ms,0,blend_radius_m)
    |   speed_ms = 0.02
    |   movel([0.097593, -1.455702, -2.509690, -0.746997, 1.570796, 1.668389],accel_mss,speed_ms,0,blend_radius_m)
    |   movel([0.099096, -1.455183, -2.510114, -0.747091, 1.570796, 1.669892],accel_mss,speed_ms,0,blend_radius_m)
    |   movel([0.100532, -1.455189, -2.510110, -0.747090, 1.570796, 1.671328],accel_mss,speed_ms,0,blend_radius_m)
    |   movel([0.101729, -1.455682, -2.509706, -0.747001, 1.570796, 1.672526],accel_mss,speed_ms,0,blend_radius_m)
    |   movel([0.102540, -1.456557, -2.508989, -0.746843, 1.570796, 1.673336],accel_mss,speed_ms,0,blend_radius_m)
    |   movel([0.102817, -1.457715, -2.508039, -0.746636, 1.570796, 1.673613],accel_mss,speed_ms,0,blend_radius_m)
    |   movel([0.102487, -1.459024, -2.506961, -0.746404, 1.570796, 1.673284],accel_mss,speed_ms,0,blend_radius_m)
    |   movel([0.101471, -1.460360, -2.505859, -0.746170, 1.570796, 1.672267],accel_mss,speed_ms,0,blend_radius_m)
    |   movel([0.100331, -1.461290, -2.505091, -0.746008, 1.570796, 1.671128],accel_mss,speed_ms,0,blend_radius_m)
    |   movel([0.099242, -1.461825, -2.504647, -0.745916, 1.570796, 1.670039],accel_mss,speed_ms,0,blend_radius_m)
    |   movel([0.098163, -1.462439, -2.504139, -0.745811, 1.570796, 1.668959],accel_mss,speed_ms,0,blend_radius_m)
    |   movel([0.097740, -1.463064, -2.503621, -0.745705, 1.570796, 1.668536],accel_mss,speed_ms,0,blend_radius_m)
    |   movel([0.097656, -1.463757, -2.503045, -0.745587, 1.570796, 1.668452],accel_mss,speed_ms,0,blend_radius_m)
    |   movel([0.097883, -1.464412, -2.502500, -0.745477, 1.570796, 1.668679],accel_mss,speed_ms,0,blend_radius_m)
    |   movel([0.098396, -1.464928, -2.502071, -0.745391, 1.570796, 1.669192],accel_mss,speed_ms,0,blend_radius_m)
    |   movel([0.099307, -1.465375, -2.501698, -0.745316, 1.570796, 1.670104],accel_mss,speed_ms,0,blend_radius_m)
    |   movel([0.100349, -1.465575, -2.501531, -0.745283, 1.570796, 1.671145],accel_mss,speed_ms,0,blend_radius_m)
    |   movel([0.101520, -1.465527, -2.501571, -0.745291, 1.570796, 1.672316],accel_mss,speed_ms,0,blend_radius_m)
    |   movel([0.102826, -1.465229, -2.501820, -0.745340, 1.570796, 1.673622],accel_mss,speed_ms,0,blend_radius_m)
    |   movel([0.104186, -1.464702, -2.502259, -0.745428, 1.570796, 1.674982],accel_mss,speed_ms,0,blend_radius_m)
    |   movel([0.105528, -1.463960, -2.502876, -0.745553, 1.570796, 1.676324],accel_mss,speed_ms,0,blend_radius_m)
    |   movel([0.106851, -1.463005, -2.503669, -0.745715, 1.570796, 1.677647],accel_mss,speed_ms,0,blend_radius_m)
    |   movel([0.108159, -1.461834, -2.504640, -0.745915, 1.570796, 1.678955],accel_mss,speed_ms,0,blend_radius_m)
    |   movel([0.109978, -1.459624, -2.506467, -0.746298, 1.570796, 1.680775],accel_mss,speed_ms,0,blend_radius_m)
    |   movel([0.111097, -1.457268, -2.508406, -0.746715, 1.570796, 1.681894],accel_mss,speed_ms,0,blend_radius_m)
    |   movel([0.111370, -1.456051, -2.509404, -0.746934, 1.570796, 1.682166],accel_mss,speed_ms,0,blend_radius_m)
    |   movel([0.111419, -1.454832, -2.510402, -0.747155, 1.570796, 1.682215],accel_mss,speed_ms,0,blend_radius_m)
    |   movel([0.110851, -1.452380, -2.512401, -0.747608, 1.570796, 1.681647],accel_mss,speed_ms,0,blend_radius_m)
    |   movel([0.109332, -1.450009, -2.514327, -0.748054, 1.570796, 1.680128],accel_mss,speed_ms,0,blend_radius_m)
    |   movel([0.106804, -1.447822, -2.516095, -0.748473, 1.570796, 1.677600],accel_mss,speed_ms,0,blend_radius_m)
    |   movel([0.117518, -1.437224, -2.524559, -0.750606, 1.570796, 1.688314],accel_mss,speed_ms,0,blend_radius_m)
    |   movel([0.129939, -1.446214, -2.517390, -0.748785, 1.570796, 1.700735],accel_mss,speed_ms,0,blend_radius_m)
    |   movel([0.122923, -1.452995, -2.511901, -0.747493, 1.570796, 1.693720],accel_mss,speed_ms,0,blend_radius_m)
    |   movel([0.124124, -1.451038, -2.513492, -0.747859, 1.570796, 1.694920],accel_mss,speed_ms,0,blend_radius_m)
    |   movel([0.124786, -1.448938, -2.515193, -0.748258, 1.570796, 1.695582],accel_mss,speed_ms,0,blend_radius_m)
    |   movel([0.124868, -1.446802, -2.516916, -0.748671, 1.570796, 1.695664],accel_mss,speed_ms,0,blend_radius_m)
    |   movel([0.124338, -1.444736, -2.518577, -0.749076, 1.570796, 1.695134],accel_mss,speed_ms,0,blend_radius_m)
    |   movel([0.123179, -1.442832, -2.520101, -0.749456, 1.570796, 1.693975],accel_mss,speed_ms,0,blend_radius_m)
    |   movel([0.121391, -1.441187, -2.521413, -0.749789, 1.570796, 1.692187],accel_mss,speed_ms,0,blend_radius_m)
    |   movel([0.113466, -1.448957, -2.515177, -0.748254, 1.570796, 1.684263],accel_mss,speed_ms,0,blend_radius_m)
    |   movel([0.115713, -1.450913, -2.513593, -0.747883, 1.570796, 1.686509],accel_mss,speed_ms,0,blend_radius_m)
    |   movel([0.117412, -1.453222, -2.511716, -0.747451, 1.570796, 1.688208],accel_mss,speed_ms,0,blend_radius_m)
    |   movel([0.118379, -1.455789, -2.509619, -0.746981, 1.570796, 1.689175],accel_mss,speed_ms,0,blend_radius_m)
    |   movel([0.118524, -1.457134, -2.508515, -0.746739, 1.570796, 1.689320],accel_mss,speed_ms,0,blend_radius_m)
    |   movel([0.118441, -1.458524, -2.507373, -0.746492, 1.570796, 1.689238],accel_mss,speed_ms,0,blend_radius_m)
    |   movel([0.118097, -1.459926, -2.506218, -0.746245, 1.570796, 1.688893],accel_mss,speed_ms,0,blend_radius_m)
    |   movel([0.117452, -1.461313, -2.505072, -0.746004, 1.570796, 1.688248],accel_mss,speed_ms,0,blend_radius_m)
    |   movel([0.116509, -1.462686, -2.503934, -0.745769, 1.570796, 1.687305],accel_mss,speed_ms,0,blend_radius_m)
    |   movel([0.115268, -1.464045, -2.502805, -0.745539, 1.570796, 1.686064],accel_mss,speed_ms,0,blend_radius_m)
    |   movel([0.113855, -1.465280, -2.501777, -0.745332, 1.570796, 1.684652],accel_mss,speed_ms,0,blend_radius_m)
    |   movel([0.112394, -1.466285, -2.500939, -0.745165, 1.570796, 1.683190],accel_mss,speed_ms,0,blend_radius_m)
    |   movel([0.110882, -1.467060, -2.500292, -0.745038, 1.570796, 1.681679],accel_mss,speed_ms,0,blend_radius_m)
    |   movel([0.109317, -1.467606, -2.499835, -0.744949, 1.570796, 1.680114],accel_mss,speed_ms,0,blend_radius_m)
    |   movel([0.106199, -1.468111, -2.499411, -0.744867, 1.570796, 1.676996],accel_mss,speed_ms,0,blend_radius_m)
    |   movel([0.103209, -1.467898, -2.499590, -0.744901, 1.570796, 1.674005],accel_mss,speed_ms,0,blend_radius_m)
    |   movel([0.100457, -1.467096, -2.500261, -0.745032, 1.570796, 1.671254],accel_mss,speed_ms,0,blend_radius_m)
    |   movel([0.098069, -1.465832, -2.501317, -0.745240, 1.570796, 1.668865],accel_mss,speed_ms,0,blend_radius_m)
    |   movel([0.096712, -1.464684, -2.502274, -0.745431, 1.570796, 1.667508],accel_mss,speed_ms,0,blend_radius_m)
    |   movel([0.095606, -1.463254, -2.503463, -0.745672, 1.570796, 1.666403],accel_mss,speed_ms,0,blend_radius_m)
    |   movel([0.094883, -1.461644, -2.504797, -0.745947, 1.570796, 1.665679],accel_mss,speed_ms,0,blend_radius_m)
    |   movel([0.094684, -1.459957, -2.506192, -0.746240, 1.570796, 1.665481],accel_mss,speed_ms,0,blend_radius_m)
    |   movel([0.095089, -1.458302, -2.507556, -0.746531, 1.570796, 1.665886],accel_mss,speed_ms,0,blend_radius_m)
    |   movel([0.096184, -1.456785, -2.508802, -0.746802, 1.570796, 1.666981],accel_mss,speed_ms,0,blend_radius_m)
    |   speed_ms = 0.003
    |   movel([0.096184, -1.450724, -2.506032, -0.755633, 1.570796, 1.666981],accel_mss,speed_ms,0,blend_radius_m)
    |   speed_ms = 0.05
    |   movel([0.096184, -1.427284, -2.494664, -0.790441, 1.570796, 1.666981],accel_mss,speed_ms,0,blend_radius_m)
    |   #M_RunCode9
    |   movel([0.065363, -1.369061, -2.537910, -0.805417, 1.570796, 1.636159],accel_mss,speed_ms,0,blend_radius_m)
    |   #M_RunCode3
    |   movel([0.065363, -1.393636, -2.549996, -0.768757, 1.570796, 1.636159],accel_mss,speed_ms,0,blend_radius_m)
    |   speed_ms = 0.003
    |   movel([0.065363, -1.400012, -2.552945, -0.759432, 1.570796, 1.636159],accel_mss,speed_ms,0,blend_radius_m)
    |   speed_ms = 0.02
    |   movel([0.062779, -1.401414, -2.551912, -0.759062, 1.570796, 1.633576],accel_mss,speed_ms,0,blend_radius_m)
    |   movel([0.060012, -1.402408, -2.551179, -0.758802, 1.570796, 1.630808],accel_mss,speed_ms,0,blend_radius_m)
    |   movel([0.057163, -1.403040, -2.550712, -0.758637, 1.570796, 1.627959],accel_mss,speed_ms,0,blend_radius_m)
    |   movel([0.054336, -1.403351, -2.550482, -0.758556, 1.570796, 1.625132],accel_mss,speed_ms,0,blend_radius_m)
    |   movel([0.051638, -1.403378, -2.550462, -0.758549, 1.570796, 1.622434],accel_mss,speed_ms,0,blend_radius_m)
    |   movel([0.051705, -1.400681, -2.552453, -0.759255, 1.570796, 1.622501],accel_mss,speed_ms,0,blend_radius_m)
    |   movel([0.052593, -1.397500, -2.554788, -0.760101, 1.570796, 1.623390],accel_mss,speed_ms,0,blend_radius_m)
    |   movel([0.054194, -1.394122, -2.557251, -0.761016, 1.570796, 1.624991],accel_mss,speed_ms,0,blend_radius_m)
    |   movel([0.056383, -1.390860, -2.559614, -0.761915, 1.570796, 1.627180],accel_mss,speed_ms,0,blend_radius_m)
    |   movel([0.059042, -1.388022, -2.561657, -0.762710, 1.570796, 1.629838],accel_mss,speed_ms,0,blend_radius_m)
    |   movel([0.060505, -1.386862, -2.562489, -0.763038, 1.570796, 1.631301],accel_mss,speed_ms,0,blend_radius_m)
    |   movel([0.062034, -1.385928, -2.563158, -0.763304, 1.570796, 1.632830],accel_mss,speed_ms,0,blend_radius_m)
    |   movel([0.063614, -1.385260, -2.563635, -0.763495, 1.570796, 1.634411],accel_mss,speed_ms,0,blend_radius_m)
    |   movel([0.065228, -1.384898, -2.563893, -0.763598, 1.570796, 1.636025],accel_mss,speed_ms,0,blend_radius_m)
    |   movel([0.066855, -1.384880, -2.563906, -0.763603, 1.570796, 1.637651],accel_mss,speed_ms,0,blend_radius_m)
    |   movel([0.068475, -1.385252, -2.563640, -0.763497, 1.570796, 1.639272],accel_mss,speed_ms,0,blend_radius_m)
    |   movel([0.070360, -1.386422, -2.562804, -0.763163, 1.570796, 1.641156],accel_mss,speed_ms,0,blend_radius_m)
    |   movel([0.071352, -1.388167, -2.561553, -0.762669, 1.570796, 1.642148],accel_mss,speed_ms,0,blend_radius_m)
    |   movel([0.071524, -1.390371, -2.559967, -0.762051, 1.570796, 1.642320],accel_mss,speed_ms,0,blend_radius_m)
    |   movel([0.070946, -1.392916, -2.558126, -0.761347, 1.570796, 1.641743],accel_mss,speed_ms,0,blend_radius_m)
    |   movel([0.069554, -1.395810, -2.556022, -0.760557, 1.570796, 1.640350],accel_mss,speed_ms,0,blend_radius_m)
    |   movel([0.067656, -1.398159, -2.554305, -0.759925, 1.570796, 1.638453],accel_mss,speed_ms,0,blend_radius_m)
    |   movel([0.065363, -1.400012, -2.552945, -0.759432, 1.570796, 1.636159],accel_mss,speed_ms,0,blend_radius_m)
    |   speed_ms = 0.003
    |   movel([0.065363, -1.393636, -2.549996, -0.768757, 1.570796, 1.636159],accel_mss,speed_ms,0,blend_radius_m)
    |   speed_ms = 0.05
    |   movel([0.065363, -1.369061, -2.537910, -0.805417, 1.570796, 1.636159],accel_mss,speed_ms,0,blend_radius_m)
    |   #M_RunCode9
    |   movel([0.108201, -1.279960, -2.595203, -0.837226, 1.570796, 1.678998],accel_mss,speed_ms,0,blend_radius_m)
    |   #M_RunCode3
    |   movel([0.108201, -1.306030, -2.608435, -0.797923, 1.570796, 1.678998],accel_mss,speed_ms,0,blend_radius_m)
    |   speed_ms = 0.003
    |   movel([0.108201, -1.312833, -2.611673, -0.787882, 1.570796, 1.678998],accel_mss,speed_ms,0,blend_radius_m)
    |   speed_ms = 0.02
    |   movel([0.106517, -1.312610, -2.611810, -0.787968, 1.570796, 1.677313],accel_mss,speed_ms,0,blend_radius_m)
    |   movel([0.105092, -1.311943, -2.612220, -0.788226, 1.570796, 1.675888],accel_mss,speed_ms,0,blend_radius_m)
    |   movel([0.103827, -1.311038, -2.612774, -0.788577, 1.570796, 1.674623],accel_mss,speed_ms,0,blend_radius_m)
    |   movel([0.104560, -1.310549, -2.613073, -0.788767, 1.570796, 1.675356],accel_mss,speed_ms,0,blend_radius_m)
    |   movel([0.105215, -1.310555, -2.613069, -0.788765, 1.570796, 1.676012],accel_mss,speed_ms,0,blend_radius_m)
    |   movel([0.105997, -1.310511, -2.613096, -0.788782, 1.570796, 1.676793],accel_mss,speed_ms,0,blend_radius_m)
    |   movel([0.107100, -1.309876, -2.613484, -0.789029, 1.570796, 1.677896],accel_mss,speed_ms,0,blend_radius_m)
    |   movel([0.108084, -1.308861, -2.614103, -0.789425, 1.570796, 1.678880],accel_mss,speed_ms,0,blend_radius_m)
    |   movel([0.108901, -1.307727, -2.614792, -0.789870, 1.570796, 1.679697],accel_mss,speed_ms,0,blend_radius_m)
    |   movel([0.109984, -1.306129, -2.615761, -0.790499, 1.570796, 1.680780],accel_mss,speed_ms,0,blend_radius_m)
    |   movel([0.108500, -1.304879, -2.616517, -0.790993, 1.570796, 1.679297],accel_mss,speed_ms,0,blend_radius_m)
    |   movel([0.106768, -1.304387, -2.616814, -0.791188, 1.570796, 1.677564],accel_mss,speed_ms,0,blend_radius_m)
    |   movel([0.105805, -1.304516, -2.616736, -0.791137, 1.570796, 1.676602],accel_mss,speed_ms,0,blend_radius_m)
    |   movel([0.104779, -1.304946, -2.616477, -0.790967, 1.570796, 1.675575],accel_mss,speed_ms,0,blend_radius_m)
    |   movel([0.103687, -1.305712, -2.616013, -0.790663, 1.570796, 1.674483],accel_mss,speed_ms,0,blend_radius_m)
    |   movel([0.102532, -1.306852, -2.615323, -0.790214, 1.570796, 1.673328],accel_mss,speed_ms,0,blend_radius_m)
    |   movel([0.102352, -1.305645, -2.616054, -0.790690, 1.570796, 1.673149],accel_mss,speed_ms,0,blend_radius_m)
    |   movel([0.102385, -1.304530, -2.616728, -0.791132, 1.570796, 1.673181],accel_mss,speed_ms,0,blend_radius_m)
    |   movel([0.102578, -1.304058, -2.617012, -0.791319, 1.570796, 1.673375],accel_mss,speed_ms,0,blend_radius_m)
    |   movel([0.102946, -1.303674, -2.617244, -0.791472, 1.570796, 1.673743],accel_mss,speed_ms,0,blend_radius_m)
    |   movel([0.104357, -1.303249, -2.617500, -0.791641, 1.570796, 1.675154],accel_mss,speed_ms,0,blend_radius_m)
    |   movel([0.107054, -1.303315, -2.617459, -0.791614, 1.570796, 1.677851],accel_mss,speed_ms,0,blend_radius_m)
    |   movel([0.109447, -1.304023, -2.617034, -0.791333, 1.570796, 1.680243],accel_mss,speed_ms,0,blend_radius_m)
    |   movel([0.110353, -1.304653, -2.616653, -0.791083, 1.570796, 1.681150],accel_mss,speed_ms,0,blend_radius_m)
    |   movel([0.110971, -1.305491, -2.616147, -0.790751, 1.570796, 1.681767],accel_mss,speed_ms,0,blend_radius_m)
    |   movel([0.111233, -1.306548, -2.615508, -0.790334, 1.570796, 1.682029],accel_mss,speed_ms,0,blend_radius_m)
    |   movel([0.111068, -1.307839, -2.614724, -0.789826, 1.570796, 1.681865],accel_mss,speed_ms,0,blend_radius_m)
    |   movel([0.109348, -1.307847, -2.614720, -0.789823, 1.570796, 1.680145],accel_mss,speed_ms,0,blend_radius_m)
    |   movel([0.110243, -1.312399, -2.611940, -0.788050, 1.570796, 1.681040],accel_mss,speed_ms,0,blend_radius_m)
    |   movel([0.108201, -1.312833, -2.611673, -0.787882, 1.570796, 1.678998],accel_mss,speed_ms,0,blend_radius_m)
    |   speed_ms = 0.003
    |   movel([0.108201, -1.306030, -2.608435, -0.797923, 1.570796, 1.678998],accel_mss,speed_ms,0,blend_radius_m)
    |   speed_ms = 0.05
    |   movel([0.108201, -1.279960, -2.595203, -0.837226, 1.570796, 1.678998],accel_mss,speed_ms,0,blend_radius_m)
    |   #M_RunCode9
    |   movel([0.068183, -1.263928, -2.604442, -0.844019, 1.570796, 1.638979],accel_mss,speed_ms,0,blend_radius_m)
    |   #M_RunCode3
    |   movel([0.068183, -1.290226, -2.617885, -0.804278, 1.570796, 1.638979],accel_mss,speed_ms,0,blend_radius_m)
    |   speed_ms = 0.003
    |   movel([0.068183, -1.297097, -2.621176, -0.794116, 1.570796, 1.638979],accel_mss,speed_ms,0,blend_radius_m)
    |   speed_ms = 0.02
    |   movel([0.066467, -1.299361, -2.619829, -0.793200, 1.570796, 1.637264],accel_mss,speed_ms,0,blend_radius_m)
    |   movel([0.064519, -1.301543, -2.618524, -0.792322, 1.570796, 1.635316],accel_mss,speed_ms,0,blend_radius_m)
    |   movel([0.062350, -1.303607, -2.617284, -0.791498, 1.570796, 1.633146],accel_mss,speed_ms,0,blend_radius_m)
    |   movel([0.059974, -1.305526, -2.616126, -0.790737, 1.570796, 1.630771],accel_mss,speed_ms,0,blend_radius_m)
    |   movel([0.057413, -1.307268, -2.615071, -0.790050, 1.570796, 1.628210],accel_mss,speed_ms,0,blend_radius_m)
    |   movel([0.055975, -1.307970, -2.614644, -0.789774, 1.570796, 1.626771],accel_mss,speed_ms,0,blend_radius_m)
    |   movel([0.054432, -1.308529, -2.614305, -0.789555, 1.570796, 1.625229],accel_mss,speed_ms,0,blend_radius_m)
    |   movel([0.053046, -1.309040, -2.613993, -0.789355, 1.570796, 1.623842],accel_mss,speed_ms,0,blend_radius_m)
    |   movel([0.052086, -1.309587, -2.613660, -0.789142, 1.570796, 1.622882],accel_mss,speed_ms,0,blend_radius_m)
    |   movel([0.050909, -1.311045, -2.612770, -0.788574, 1.570796, 1.621705],accel_mss,speed_ms,0,blend_radius_m)
    |   movel([0.049542, -1.313173, -2.611465, -0.787751, 1.570796, 1.620338],accel_mss,speed_ms,0,blend_radius_m)
    |   movel([0.048143, -1.315401, -2.610092, -0.786896, 1.570796, 1.618940],accel_mss,speed_ms,0,blend_radius_m)
    |   movel([0.046861, -1.317165, -2.609001, -0.786223, 1.570796, 1.617657],accel_mss,speed_ms,0,blend_radius_m)
    |   movel([0.043920, -1.320192, -2.607119, -0.785078, 1.570796, 1.614716],accel_mss,speed_ms,0,blend_radius_m)
    |   movel([0.041006, -1.322557, -2.605639, -0.784192, 1.570796, 1.611803],accel_mss,speed_ms,0,blend_radius_m)
    |   movel([0.038118, -1.324329, -2.604527, -0.783534, 1.570796, 1.608914],accel_mss,speed_ms,0,blend_radius_m)
    |   movel([0.035257, -1.325566, -2.603747, -0.783076, 1.570796, 1.606054],accel_mss,speed_ms,0,blend_radius_m)
    |   movel([0.032430, -1.326331, -2.603264, -0.782794, 1.570796, 1.603226],accel_mss,speed_ms,0,blend_radius_m)
    |   movel([0.029639, -1.326680, -2.603043, -0.782666, 1.570796, 1.600436],accel_mss,speed_ms,0,blend_radius_m)
    |   movel([0.026891, -1.326669, -2.603050, -0.782670, 1.570796, 1.597687],accel_mss,speed_ms,0,blend_radius_m)
    |   movel([0.024187, -1.326357, -2.603248, -0.782785, 1.570796, 1.594984],accel_mss,speed_ms,0,blend_radius_m)
    |   movel([0.018950, -1.325045, -2.604075, -0.783268, 1.570796, 1.589746],accel_mss,speed_ms,0,blend_radius_m)
    |   movel([0.013993, -1.323179, -2.605249, -0.783961, 1.570796, 1.584790],accel_mss,speed_ms,0,blend_radius_m)
    |   movel([0.005237, -1.319507, -2.607546, -0.785336, 1.570796, 1.576034],accel_mss,speed_ms,0,blend_radius_m)
    |   movel([0.001064, -1.318336, -2.608275, -0.785779, 1.570796, 1.571861],accel_mss,speed_ms,0,blend_radius_m)
    |   movel([-0.004062, -1.317433, -2.608835, -0.786121, 1.570796, 1.566734],accel_mss,speed_ms,0,blend_radius_m)
    |   movel([-0.009890, -1.316882, -2.609177, -0.786331, 1.570796, 1.560907],accel_mss,speed_ms,0,blend_radius_m)
    |   movel([-0.016155, -1.316757, -2.609254, -0.786378, 1.570796, 1.554641],accel_mss,speed_ms,0,blend_radius_m)
    |   movel([-0.022589, -1.317129, -2.609023, -0.786237, 1.570796, 1.548207],accel_mss,speed_ms,0,blend_radius_m)
    |   movel([-0.028918, -1.318053, -2.608450, -0.785886, 1.570796, 1.541878],accel_mss,speed_ms,0,blend_radius_m)
    |   movel([-0.034863, -1.319579, -2.607501, -0.785309, 1.570796, 1.535934],accel_mss,speed_ms,0,blend_radius_m)
    |   movel([-0.037604, -1.320583, -2.606874, -0.784931, 1.570796, 1.533193],accel_mss,speed_ms,0,blend_radius_m)
    |   movel([-0.040145, -1.321751, -2.606144, -0.784493, 1.570796, 1.530652],accel_mss,speed_ms,0,blend_radius_m)
    |   movel([-0.042700, -1.323193, -2.605240, -0.783955, 1.570796, 1.528096],accel_mss,speed_ms,0,blend_radius_m)
    |   movel([-0.045606, -1.325084, -2.604051, -0.783254, 1.570796, 1.525190],accel_mss,speed_ms,0,blend_radius_m)
    |   movel([-0.048654, -1.327357, -2.602615, -0.782417, 1.570796, 1.522142],accel_mss,speed_ms,0,blend_radius_m)
    |   movel([-0.051646, -1.329942, -2.600973, -0.781474, 1.570796, 1.519150],accel_mss,speed_ms,0,blend_radius_m)
    |   movel([-0.054374, -1.332764, -2.599170, -0.780455, 1.570796, 1.516423],accel_mss,speed_ms,0,blend_radius_m)
    |   movel([-0.056644, -1.335756, -2.597247, -0.779386, 1.570796, 1.514152],accel_mss,speed_ms,0,blend_radius_m)
    |   movel([-0.058260, -1.338847, -2.595248, -0.778294, 1.570796, 1.512537],accel_mss,speed_ms,0,blend_radius_m)
    |   movel([-0.058764, -1.340407, -2.594234, -0.777748, 1.570796, 1.512032],accel_mss,speed_ms,0,blend_radius_m)
    |   movel([-0.059032, -1.341968, -2.593216, -0.777205, 1.570796, 1.511764],accel_mss,speed_ms,0,blend_radius_m)
    |   movel([-0.058880, -1.344184, -2.591765, -0.776440, 1.570796, 1.511916],accel_mss,speed_ms,0,blend_radius_m)
    |   movel([-0.058008, -1.345772, -2.590721, -0.775896, 1.570796, 1.512788],accel_mss,speed_ms,0,blend_radius_m)
    |   movel([-0.056501, -1.346799, -2.590044, -0.775545, 1.570796, 1.514295],accel_mss,speed_ms,0,blend_radius_m)
    |   movel([-0.054442, -1.347330, -2.589694, -0.775365, 1.570796, 1.516354],accel_mss,speed_ms,0,blend_radius_m)
    |   movel([-0.051910, -1.347426, -2.589630, -0.775332, 1.570796, 1.518886],accel_mss,speed_ms,0,blend_radius_m)
    |   movel([-0.048987, -1.347151, -2.589812, -0.775426, 1.570796, 1.521810],accel_mss,speed_ms,0,blend_radius_m)
    |   movel([-0.045747, -1.346563, -2.590200, -0.775626, 1.570796, 1.525049],accel_mss,speed_ms,0,blend_radius_m)
    |   movel([-0.042271, -1.345725, -2.590752, -0.775912, 1.570796, 1.528526],accel_mss,speed_ms,0,blend_radius_m)
    |   movel([-0.034933, -1.343530, -2.592194, -0.776665, 1.570796, 1.535863],accel_mss,speed_ms,0,blend_radius_m)
    |   movel([-0.027609, -1.341035, -2.593825, -0.777529, 1.570796, 1.543188],accel_mss,speed_ms,0,blend_radius_m)
    |   movel([-0.020959, -1.338699, -2.595344, -0.778346, 1.570796, 1.549838],accel_mss,speed_ms,0,blend_radius_m)
    |   movel([-0.015651, -1.336987, -2.596453, -0.778949, 1.570796, 1.555145],accel_mss,speed_ms,0,blend_radius_m)
    |   movel([-0.002809, -1.333318, -2.598815, -0.780256, 1.570796, 1.567988],accel_mss,speed_ms,0,blend_radius_m)
    |   movel([0.004059, -1.331537, -2.599955, -0.780897, 1.570796, 1.574855],accel_mss,speed_ms,0,blend_radius_m)
    |   movel([0.009383, -1.330453, -2.600647, -0.781289, 1.570796, 1.580179],accel_mss,speed_ms,0,blend_radius_m)
    |   movel([0.011398, -1.330291, -2.600751, -0.781348, 1.570796, 1.582194],accel_mss,speed_ms,0,blend_radius_m)
    |   movel([0.013270, -1.330370, -2.600700, -0.781319, 1.570796, 1.584066],accel_mss,speed_ms,0,blend_radius_m)
    |   movel([0.016577, -1.331200, -2.600171, -0.781018, 1.570796, 1.587373],accel_mss,speed_ms,0,blend_radius_m)
    |   movel([0.019297, -1.332810, -2.599141, -0.780438, 1.570796, 1.590093],accel_mss,speed_ms,0,blend_radius_m)
    |   movel([0.021435, -1.335056, -2.597698, -0.779635, 1.570796, 1.592231],accel_mss,speed_ms,0,blend_radius_m)
    |   movel([0.022985, -1.337804, -2.595924, -0.778661, 1.570796, 1.593781],accel_mss,speed_ms,0,blend_radius_m)
    |   movel([0.023955, -1.340917, -2.593902, -0.777570, 1.570796, 1.594751],accel_mss,speed_ms,0,blend_radius_m)
    |   movel([0.024352, -1.344258, -2.591716, -0.776414, 1.570796, 1.595148],accel_mss,speed_ms,0,blend_radius_m)
    |   movel([0.024181, -1.347692, -2.589455, -0.775242, 1.570796, 1.594978],accel_mss,speed_ms,0,blend_radius_m)
    |   movel([0.023212, -1.352030, -2.586574, -0.773785, 1.570796, 1.594008],accel_mss,speed_ms,0,blend_radius_m)
    |   movel([0.022491, -1.353877, -2.585340, -0.773172, 1.570796, 1.593287],accel_mss,speed_ms,0,blend_radius_m)
    |   movel([0.021617, -1.355544, -2.584222, -0.772623, 1.570796, 1.592413],accel_mss,speed_ms,0,blend_radius_m)
    |   movel([0.020604, -1.357053, -2.583206, -0.772130, 1.570796, 1.591400],accel_mss,speed_ms,0,blend_radius_m)
    |   movel([0.019454, -1.358428, -2.582278, -0.771683, 1.570796, 1.590251],accel_mss,speed_ms,0,blend_radius_m)
    |   movel([0.016782, -1.360879, -2.580617, -0.770893, 1.570796, 1.587578],accel_mss,speed_ms,0,blend_radius_m)
    |   movel([0.013656, -1.363086, -2.579115, -0.770188, 1.570796, 1.584452],accel_mss,speed_ms,0,blend_radius_m)
    |   movel([0.010137, -1.365236, -2.577644, -0.769509, 1.570796, 1.580933],accel_mss,speed_ms,0,blend_radius_m)
    |   movel([0.002163, -1.370091, -2.574300, -0.767998, 1.570796, 1.572959],accel_mss,speed_ms,0,blend_radius_m)
    |   movel([0.001770, -1.370367, -2.574108, -0.767913, 1.570796, 1.572566],accel_mss,speed_ms,0,blend_radius_m)
    |   movel([0.001962, -1.370367, -2.574109, -0.767914, 1.570796, 1.572759],accel_mss,speed_ms,0,blend_radius_m)
    |   movel([0.003797, -1.369678, -2.574586, -0.768126, 1.570796, 1.574594],accel_mss,speed_ms,0,blend_radius_m)
    |   movel([0.011160, -1.366566, -2.576731, -0.769092, 1.570796, 1.581956],accel_mss,speed_ms,0,blend_radius_m)
    |   movel([0.023447, -1.361411, -2.580256, -0.770722, 1.570796, 1.594243],accel_mss,speed_ms,0,blend_radius_m)
    |   movel([0.017685, -1.366383, -2.576857, -0.769149, 1.570796, 1.588482],accel_mss,speed_ms,0,blend_radius_m)
    |   movel([0.011119, -1.371663, -2.573210, -0.767516, 1.570796, 1.581916],accel_mss,speed_ms,0,blend_radius_m)
    |   movel([0.004025, -1.377088, -2.569421, -0.765880, 1.570796, 1.574821],accel_mss,speed_ms,0,blend_radius_m)
    |   movel([-0.003343, -1.382493, -2.565605, -0.764291, 1.570796, 1.567454],accel_mss,speed_ms,0,blend_radius_m)
    |   movel([-0.017889, -1.392616, -2.558343, -0.761429, 1.570796, 1.552908],accel_mss,speed_ms,0,blend_radius_m)
    |   movel([-0.024590, -1.397017, -2.555141, -0.760231, 1.570796, 1.546206],accel_mss,speed_ms,0,blend_radius_m)
    |   movel([-0.030606, -1.400773, -2.552385, -0.759231, 1.570796, 1.540190],accel_mss,speed_ms,0,blend_radius_m)
    |   movel([-0.037332, -1.408268, -2.546824, -0.757297, 1.570796, 1.533464],accel_mss,speed_ms,0,blend_radius_m)
    |   movel([-0.043886, -1.416131, -2.540902, -0.755356, 1.570796, 1.526910],accel_mss,speed_ms,0,blend_radius_m)
    |   movel([-0.056627, -1.432235, -2.528484, -0.751670, 1.570796, 1.514169],accel_mss,speed_ms,0,blend_radius_m)
    |   movel([-0.062904, -1.440143, -2.522245, -0.750002, 1.570796, 1.507892],accel_mss,speed_ms,0,blend_radius_m)
    |   movel([-0.069187, -1.447749, -2.516153, -0.748487, 1.570796, 1.501610],accel_mss,speed_ms,0,blend_radius_m)
    |   movel([-0.075526, -1.454908, -2.510340, -0.747142, 1.570796, 1.495270],accel_mss,speed_ms,0,blend_radius_m)
    |   movel([-0.081984, -1.461480, -2.504933, -0.745976, 1.570796, 1.488813],accel_mss,speed_ms,0,blend_radius_m)
    |   movel([-0.084611, -1.463841, -2.502975, -0.745573, 1.570796, 1.486186],accel_mss,speed_ms,0,blend_radius_m)
    |   movel([-0.087222, -1.465905, -2.501256, -0.745228, 1.570796, 1.483574],accel_mss,speed_ms,0,blend_radius_m)
    |   movel([-0.089796, -1.467667, -2.499783, -0.744939, 1.570796, 1.481000],accel_mss,speed_ms,0,blend_radius_m)
    |   movel([-0.092315, -1.469128, -2.498559, -0.744703, 1.570796, 1.478481],accel_mss,speed_ms,0,blend_radius_m)
    |   movel([-0.094761, -1.470280, -2.497591, -0.744519, 1.570796, 1.476035],accel_mss,speed_ms,0,blend_radius_m)
    |   movel([-0.097118, -1.471120, -2.496884, -0.744386, 1.570796, 1.473678],accel_mss,speed_ms,0,blend_radius_m)
    |   movel([-0.099367, -1.471645, -2.496441, -0.744303, 1.570796, 1.471430],accel_mss,speed_ms,0,blend_radius_m)
    |   movel([-0.101485, -1.471850, -2.496268, -0.744271, 1.570796, 1.469311],accel_mss,speed_ms,0,blend_radius_m)
    |   movel([-0.103458, -1.471728, -2.496371, -0.744290, 1.570796, 1.467338],accel_mss,speed_ms,0,blend_radius_m)
    |   movel([-0.105267, -1.471271, -2.496756, -0.744362, 1.570796, 1.465529],accel_mss,speed_ms,0,blend_radius_m)
    |   movel([-0.106888, -1.470476, -2.497426, -0.744487, 1.570796, 1.463908],accel_mss,speed_ms,0,blend_radius_m)
    |   movel([-0.108306, -1.469335, -2.498385, -0.744669, 1.570796, 1.462490],accel_mss,speed_ms,0,blend_radius_m)
    |   movel([-0.109498, -1.467837, -2.499641, -0.744911, 1.570796, 1.461298],accel_mss,speed_ms,0,blend_radius_m)
    |   movel([-0.110443, -1.465975, -2.501198, -0.745216, 1.570796, 1.460354],accel_mss,speed_ms,0,blend_radius_m)
    |   movel([-0.111118, -1.463738, -2.503060, -0.745590, 1.570796, 1.459678],accel_mss,speed_ms,0,blend_radius_m)
    |   movel([-0.111501, -1.461116, -2.505234, -0.746038, 1.570796, 1.459295],accel_mss,speed_ms,0,blend_radius_m)
    |   movel([-0.108428, -1.460890, -2.505421, -0.746077, 1.570796, 1.462368],accel_mss,speed_ms,0,blend_radius_m)
    |   movel([-0.106908, -1.460703, -2.505576, -0.746110, 1.570796, 1.463888],accel_mss,speed_ms,0,blend_radius_m)
    |   movel([-0.105411, -1.460222, -2.505973, -0.746194, 1.570796, 1.465385],accel_mss,speed_ms,0,blend_radius_m)
    |   movel([-0.104290, -1.459531, -2.506543, -0.746314, 1.570796, 1.466507],accel_mss,speed_ms,0,blend_radius_m)
    |   movel([-0.103032, -1.458465, -2.507421, -0.746502, 1.570796, 1.467764],accel_mss,speed_ms,0,blend_radius_m)
    |   movel([-0.100191, -1.455393, -2.509943, -0.747053, 1.570796, 1.470605],accel_mss,speed_ms,0,blend_radius_m)
    |   movel([-0.097046, -1.451378, -2.513216, -0.747795, 1.570796, 1.473751],accel_mss,speed_ms,0,blend_radius_m)
    |   movel([-0.093767, -1.446796, -2.516921, -0.748672, 1.570796, 1.477029],accel_mss,speed_ms,0,blend_radius_m)
    |   movel([-0.087526, -1.437499, -2.524341, -0.750549, 1.570796, 1.483270],accel_mss,speed_ms,0,blend_radius_m)
    |   movel([-0.082980, -1.430709, -2.529678, -0.752002, 1.570796, 1.487817],accel_mss,speed_ms,0,blend_radius_m)
    |   movel([-0.078610, -1.425001, -2.534110, -0.753278, 1.570796, 1.492187],accel_mss,speed_ms,0,blend_radius_m)
    |   movel([-0.074184, -1.419247, -2.538529, -0.754613, 1.570796, 1.496612],accel_mss,speed_ms,0,blend_radius_m)
    |   movel([-0.086686, -1.425887, -2.533425, -0.753076, 1.570796, 1.484110],accel_mss,speed_ms,0,blend_radius_m)
    |   movel([-0.093236, -1.429109, -2.530925, -0.752355, 1.570796, 1.477560],accel_mss,speed_ms,0,blend_radius_m)
    |   movel([-0.099707, -1.431785, -2.528837, -0.751767, 1.570796, 1.471089],accel_mss,speed_ms,0,blend_radius_m)
    |   movel([-0.102852, -1.432803, -2.528039, -0.751547, 1.570796, 1.467944],accel_mss,speed_ms,0,blend_radius_m)
    |   movel([-0.105905, -1.433551, -2.527453, -0.751385, 1.570796, 1.464891],accel_mss,speed_ms,0,blend_radius_m)
    |   movel([-0.108844, -1.433981, -2.527115, -0.751293, 1.570796, 1.461953],accel_mss,speed_ms,0,blend_radius_m)
    |   movel([-0.111645, -1.434049, -2.527061, -0.751279, 1.570796, 1.459152],accel_mss,speed_ms,0,blend_radius_m)
    |   movel([-0.114286, -1.433710, -2.527327, -0.751351, 1.570796, 1.456511],accel_mss,speed_ms,0,blend_radius_m)
    |   movel([-0.116745, -1.432918, -2.527949, -0.751522, 1.570796, 1.454051],accel_mss,speed_ms,0,blend_radius_m)
    |   movel([-0.119001, -1.431623, -2.528964, -0.751803, 1.570796, 1.451796],accel_mss,speed_ms,0,blend_radius_m)
    |   movel([-0.121027, -1.429776, -2.530406, -0.752207, 1.570796, 1.449769],accel_mss,speed_ms,0,blend_radius_m)
    |   movel([-0.122791, -1.427103, -2.532483, -0.752802, 1.570796, 1.448006],accel_mss,speed_ms,0,blend_radius_m)
    |   movel([-0.123861, -1.423903, -2.534957, -0.753529, 1.570796, 1.446935],accel_mss,speed_ms,0,blend_radius_m)
    |   movel([-0.124248, -1.420289, -2.537732, -0.754367, 1.570796, 1.446549],accel_mss,speed_ms,0,blend_radius_m)
    |   movel([-0.123951, -1.416377, -2.540715, -0.755297, 1.570796, 1.446845],accel_mss,speed_ms,0,blend_radius_m)
    |   movel([-0.122977, -1.412289, -2.543807, -0.756293, 1.570796, 1.447819],accel_mss,speed_ms,0,blend_radius_m)
    |   movel([-0.121333, -1.408148, -2.546914, -0.757327, 1.570796, 1.449464],accel_mss,speed_ms,0,blend_radius_m)
    |   movel([-0.119022, -1.404080, -2.549941, -0.758367, 1.570796, 1.451774],accel_mss,speed_ms,0,blend_radius_m)
    |   movel([-0.116056, -1.400223, -2.552790, -0.759376, 1.570796, 1.454741],accel_mss,speed_ms,0,blend_radius_m)
    |   movel([-0.114045, -1.398412, -2.554120, -0.759857, 1.570796, 1.456752],accel_mss,speed_ms,0,blend_radius_m)
    |   movel([-0.111529, -1.396740, -2.555343, -0.760306, 1.570796, 1.459267],accel_mss,speed_ms,0,blend_radius_m)
    |   movel([-0.109294, -1.395778, -2.556046, -0.760566, 1.570796, 1.461503],accel_mss,speed_ms,0,blend_radius_m)
    |   movel([-0.108526, -1.395739, -2.556074, -0.760576, 1.570796, 1.462270],accel_mss,speed_ms,0,blend_radius_m)
    |   movel([-0.108125, -1.396091, -2.555817, -0.760481, 1.570796, 1.462671],accel_mss,speed_ms,0,blend_radius_m)
    |   movel([-0.110131, -1.397391, -2.554868, -0.760131, 1.570796, 1.460665],accel_mss,speed_ms,0,blend_radius_m)
    |   movel([-0.111735, -1.398645, -2.553949, -0.759795, 1.570796, 1.459061],accel_mss,speed_ms,0,blend_radius_m)
    |   movel([-0.112960, -1.399846, -2.553067, -0.759476, 1.570796, 1.457837],accel_mss,speed_ms,0,blend_radius_m)
    |   movel([-0.113829, -1.400985, -2.552229, -0.759175, 1.570796, 1.456968],accel_mss,speed_ms,0,blend_radius_m)
    |   movel([-0.114362, -1.402055, -2.551440, -0.758894, 1.570796, 1.456434],accel_mss,speed_ms,0,blend_radius_m)
    |   movel([-0.114582, -1.403043, -2.550710, -0.758636, 1.570796, 1.456215],accel_mss,speed_ms,0,blend_radius_m)
    |   movel([-0.114509, -1.403943, -2.550043, -0.758403, 1.570796, 1.456287],accel_mss,speed_ms,0,blend_radius_m)
    |   movel([-0.114168, -1.404749, -2.549446, -0.758194, 1.570796, 1.456628],accel_mss,speed_ms,0,blend_radius_m)
    |   movel([-0.112761, -1.406041, -2.548485, -0.757863, 1.570796, 1.458035],accel_mss,speed_ms,0,blend_radius_m)
    |   movel([-0.110534, -1.406857, -2.547877, -0.757654, 1.570796, 1.460262],accel_mss,speed_ms,0,blend_radius_m)
    |   movel([-0.107648, -1.407131, -2.547673, -0.757585, 1.570796, 1.463148],accel_mss,speed_ms,0,blend_radius_m)
    |   movel([-0.104268, -1.406801, -2.547920, -0.757669, 1.570796, 1.466529],accel_mss,speed_ms,0,blend_radius_m)
    |   movel([-0.102146, -1.406257, -2.548325, -0.757808, 1.570796, 1.468650],accel_mss,speed_ms,0,blend_radius_m)
    |   movel([-0.099580, -1.405351, -2.548999, -0.758040, 1.570796, 1.471216],accel_mss,speed_ms,0,blend_radius_m)
    |   movel([-0.093351, -1.402619, -2.551023, -0.758747, 1.570796, 1.477445],accel_mss,speed_ms,0,blend_radius_m)
    |   movel([-0.086052, -1.398962, -2.553717, -0.759711, 1.570796, 1.484744],accel_mss,speed_ms,0,blend_radius_m)
    |   movel([-0.078165, -1.394723, -2.556814, -0.760852, 1.570796, 1.492632],accel_mss,speed_ms,0,blend_radius_m)
    |   movel([-0.062617, -1.385904, -2.563175, -0.763311, 1.570796, 1.508179],accel_mss,speed_ms,0,blend_radius_m)
    |   movel([-0.050873, -1.378965, -2.568100, -0.765324, 1.570796, 1.519923],accel_mss,speed_ms,0,blend_radius_m)
    |   movel([-0.044935, -1.375432, -2.570582, -0.766375, 1.570796, 1.525861],accel_mss,speed_ms,0,blend_radius_m)
    |   movel([-0.041767, -1.373440, -2.571973, -0.766976, 1.570796, 1.529030],accel_mss,speed_ms,0,blend_radius_m)
    |   movel([-0.039446, -1.371762, -2.573141, -0.767486, 1.570796, 1.531351],accel_mss,speed_ms,0,blend_radius_m)
    |   movel([-0.038880, -1.371201, -2.573530, -0.767658, 1.570796, 1.531916],accel_mss,speed_ms,0,blend_radius_m)
    |   movel([-0.038747, -1.370840, -2.573780, -0.767768, 1.570796, 1.532049],accel_mss,speed_ms,0,blend_radius_m)
    |   movel([-0.039517, -1.370447, -2.574053, -0.767889, 1.570796, 1.531280],accel_mss,speed_ms,0,blend_radius_m)
    |   movel([-0.042420, -1.370175, -2.574241, -0.767972, 1.570796, 1.528376],accel_mss,speed_ms,0,blend_radius_m)
    |   movel([-0.045673, -1.370417, -2.574074, -0.767898, 1.570796, 1.525123],accel_mss,speed_ms,0,blend_radius_m)
    |   movel([-0.052752, -1.371238, -2.573505, -0.767646, 1.570796, 1.518045],accel_mss,speed_ms,0,blend_radius_m)
    |   movel([-0.056352, -1.371220, -2.573517, -0.767652, 1.570796, 1.514444],accel_mss,speed_ms,0,blend_radius_m)
    |   movel([-0.059849, -1.370515, -2.574006, -0.767868, 1.570796, 1.510948],accel_mss,speed_ms,0,blend_radius_m)
    |   movel([-0.061524, -1.369810, -2.574494, -0.768085, 1.570796, 1.509272],accel_mss,speed_ms,0,blend_radius_m)
    |   movel([-0.063137, -1.368821, -2.575178, -0.768390, 1.570796, 1.507659],accel_mss,speed_ms,0,blend_radius_m)
    |   movel([-0.064673, -1.367508, -2.576083, -0.768798, 1.570796, 1.506123],accel_mss,speed_ms,0,blend_radius_m)
    |   movel([-0.066120, -1.365830, -2.577237, -0.769322, 1.570796, 1.504677],accel_mss,speed_ms,0,blend_radius_m)
    |   movel([-0.067547, -1.363256, -2.578999, -0.770134, 1.570796, 1.503249],accel_mss,speed_ms,0,blend_radius_m)
    |   movel([-0.068265, -1.360413, -2.580933, -0.771042, 1.570796, 1.502531],accel_mss,speed_ms,0,blend_radius_m)
    |   movel([-0.068345, -1.357334, -2.583017, -0.772038, 1.570796, 1.502451],accel_mss,speed_ms,0,blend_radius_m)
    |   movel([-0.067861, -1.354059, -2.585218, -0.773112, 1.570796, 1.502935],accel_mss,speed_ms,0,blend_radius_m)
    |   movel([-0.066892, -1.350627, -2.587509, -0.774253, 1.570796, 1.503905],accel_mss,speed_ms,0,blend_radius_m)
    |   movel([-0.065514, -1.347082, -2.589858, -0.775449, 1.570796, 1.505283],accel_mss,speed_ms,0,blend_radius_m)
    |   movel([-0.063805, -1.343463, -2.592238, -0.776688, 1.570796, 1.506992],accel_mss,speed_ms,0,blend_radius_m)
    |   movel([-0.061847, -1.339820, -2.594616, -0.777953, 1.570796, 1.508949],accel_mss,speed_ms,0,blend_radius_m)
    |   movel([-0.057594, -1.333071, -2.598973, -0.780344, 1.570796, 1.513202],accel_mss,speed_ms,0,blend_radius_m)
    |   movel([-0.053246, -1.327365, -2.602610, -0.782415, 1.570796, 1.517550],accel_mss,speed_ms,0,blend_radius_m)
    |   movel([-0.049175, -1.322797, -2.605489, -0.784103, 1.570796, 1.521621],accel_mss,speed_ms,0,blend_radius_m)
    |   movel([-0.045759, -1.319461, -2.607574, -0.785353, 1.570796, 1.525038],accel_mss,speed_ms,0,blend_radius_m)
    |   movel([-0.040292, -1.314943, -2.610375, -0.787071, 1.570796, 1.530505],accel_mss,speed_ms,0,blend_radius_m)
    |   movel([-0.034578, -1.311061, -2.612760, -0.788568, 1.570796, 1.536218],accel_mss,speed_ms,0,blend_radius_m)
    |   movel([-0.028705, -1.307842, -2.614723, -0.789825, 1.570796, 1.542092],accel_mss,speed_ms,0,blend_radius_m)
    |   movel([-0.022770, -1.305311, -2.616256, -0.790822, 1.570796, 1.548026],accel_mss,speed_ms,0,blend_radius_m)
    |   movel([-0.016869, -1.303494, -2.617352, -0.791543, 1.570796, 1.553927],accel_mss,speed_ms,0,blend_radius_m)
    |   movel([-0.011094, -1.302405, -2.618006, -0.791977, 1.570796, 1.559702],accel_mss,speed_ms,0,blend_radius_m)
    |   movel([-0.005542, -1.302059, -2.618214, -0.792116, 1.570796, 1.565254],accel_mss,speed_ms,0,blend_radius_m)
    |   movel([-0.000305, -1.302469, -2.617968, -0.791952, 1.570796, 1.570491],accel_mss,speed_ms,0,blend_radius_m)
    |   movel([0.004062, -1.303490, -2.617354, -0.791545, 1.570796, 1.574858],accel_mss,speed_ms,0,blend_radius_m)
    |   movel([0.008143, -1.304902, -2.616503, -0.790984, 1.570796, 1.578940],accel_mss,speed_ms,0,blend_radius_m)
    |   movel([0.012105, -1.306375, -2.615612, -0.790402, 1.570796, 1.582901],accel_mss,speed_ms,0,blend_radius_m)
    |   movel([0.016121, -1.307577, -2.614883, -0.789929, 1.570796, 1.586917],accel_mss,speed_ms,0,blend_radius_m)
    |   movel([0.020367, -1.308183, -2.614515, -0.789691, 1.570796, 1.591163],accel_mss,speed_ms,0,blend_radius_m)
    |   movel([0.022631, -1.308159, -2.614530, -0.789700, 1.570796, 1.593428],accel_mss,speed_ms,0,blend_radius_m)
    |   movel([0.025020, -1.307866, -2.614708, -0.789815, 1.570796, 1.595816],accel_mss,speed_ms,0,blend_radius_m)
    |   movel([0.027558, -1.307261, -2.615075, -0.790053, 1.570796, 1.598354],accel_mss,speed_ms,0,blend_radius_m)
    |   movel([0.030268, -1.306302, -2.615657, -0.790430, 1.570796, 1.601065],accel_mss,speed_ms,0,blend_radius_m)
    |   movel([0.033180, -1.304946, -2.616477, -0.790967, 1.570796, 1.603976],accel_mss,speed_ms,0,blend_radius_m)
    |   movel([0.036316, -1.303148, -2.617560, -0.791681, 1.570796, 1.607112],accel_mss,speed_ms,0,blend_radius_m)
    |   movel([0.038953, -1.301257, -2.618695, -0.792437, 1.570796, 1.609750],accel_mss,speed_ms,0,blend_radius_m)
    |   movel([0.041005, -1.299290, -2.619871, -0.793228, 1.570796, 1.611801],accel_mss,speed_ms,0,blend_radius_m)
    |   movel([0.042502, -1.297297, -2.621057, -0.794035, 1.570796, 1.613298],accel_mss,speed_ms,0,blend_radius_m)
    |   movel([0.043487, -1.295326, -2.622225, -0.794838, 1.570796, 1.614283],accel_mss,speed_ms,0,blend_radius_m)
    |   movel([0.043990, -1.293428, -2.623345, -0.795616, 1.570796, 1.614787],accel_mss,speed_ms,0,blend_radius_m)
    |   movel([0.044048, -1.291659, -2.624386, -0.796345, 1.570796, 1.614844],accel_mss,speed_ms,0,blend_radius_m)
    |   movel([0.043697, -1.290068, -2.625317, -0.797004, 1.570796, 1.614493],accel_mss,speed_ms,0,blend_radius_m)
    |   movel([0.042975, -1.288711, -2.626109, -0.797568, 1.570796, 1.613771],accel_mss,speed_ms,0,blend_radius_m)
    |   movel([0.041918, -1.287643, -2.626731, -0.798015, 1.570796, 1.612714],accel_mss,speed_ms,0,blend_radius_m)
    |   movel([0.040564, -1.286917, -2.627153, -0.798319, 1.570796, 1.611360],accel_mss,speed_ms,0,blend_radius_m)
    |   movel([0.038953, -1.286587, -2.627344, -0.798457, 1.570796, 1.609749],accel_mss,speed_ms,0,blend_radius_m)
    |   movel([0.037125, -1.286707, -2.627275, -0.798407, 1.570796, 1.607921],accel_mss,speed_ms,0,blend_radius_m)
    |   movel([0.035121, -1.287322, -2.626918, -0.798149, 1.570796, 1.605918],accel_mss,speed_ms,0,blend_radius_m)
    |   movel([0.032988, -1.288486, -2.626240, -0.797662, 1.570796, 1.603784],accel_mss,speed_ms,0,blend_radius_m)
    |   movel([0.030765, -1.290248, -2.625212, -0.796929, 1.570796, 1.601562],accel_mss,speed_ms,0,blend_radius_m)
    |   movel([0.028498, -1.292646, -2.623806, -0.795937, 1.570796, 1.599294],accel_mss,speed_ms,0,blend_radius_m)
    |   movel([0.030387, -1.292087, -2.624134, -0.796168, 1.570796, 1.601183],accel_mss,speed_ms,0,blend_radius_m)
    |   movel([0.031938, -1.291937, -2.624222, -0.796230, 1.570796, 1.602735],accel_mss,speed_ms,0,blend_radius_m)
    |   movel([0.033115, -1.292170, -2.624085, -0.796133, 1.570796, 1.603912],accel_mss,speed_ms,0,blend_radius_m)
    |   movel([0.033889, -1.292762, -2.623738, -0.795890, 1.570796, 1.604685],accel_mss,speed_ms,0,blend_radius_m)
    |   movel([0.034224, -1.293689, -2.623191, -0.795508, 1.570796, 1.605020],accel_mss,speed_ms,0,blend_radius_m)
    |   movel([0.034090, -1.294926, -2.622462, -0.795001, 1.570796, 1.604886],accel_mss,speed_ms,0,blend_radius_m)
    |   movel([0.033458, -1.296443, -2.621564, -0.794382, 1.570796, 1.604255],accel_mss,speed_ms,0,blend_radius_m)
    |   movel([0.032296, -1.298217, -2.620510, -0.793662, 1.570796, 1.603093],accel_mss,speed_ms,0,blend_radius_m)
    |   movel([0.029774, -1.301019, -2.618837, -0.792532, 1.570796, 1.600571],accel_mss,speed_ms,0,blend_radius_m)
    |   movel([0.027083, -1.303091, -2.617594, -0.791704, 1.570796, 1.597879],accel_mss,speed_ms,0,blend_radius_m)
    |   movel([0.024287, -1.304489, -2.616753, -0.791148, 1.570796, 1.595084],accel_mss,speed_ms,0,blend_radius_m)
    |   movel([0.021467, -1.305259, -2.616288, -0.790843, 1.570796, 1.592264],accel_mss,speed_ms,0,blend_radius_m)
    |   movel([0.018691, -1.305446, -2.616174, -0.790769, 1.570796, 1.589488],accel_mss,speed_ms,0,blend_radius_m)
    |   movel([0.016035, -1.305094, -2.616387, -0.790908, 1.570796, 1.586831],accel_mss,speed_ms,0,blend_radius_m)
    |   movel([0.013576, -1.304241, -2.616902, -0.791246, 1.570796, 1.584373],accel_mss,speed_ms,0,blend_radius_m)
    |   movel([0.011389, -1.302930, -2.617691, -0.791768, 1.570796, 1.582186],accel_mss,speed_ms,0,blend_radius_m)
    |   movel([0.009557, -1.301188, -2.618736, -0.792464, 1.570796, 1.580353],accel_mss,speed_ms,0,blend_radius_m)
    |   movel([0.008155, -1.299061, -2.620007, -0.793320, 1.570796, 1.578952],accel_mss,speed_ms,0,blend_radius_m)
    |   movel([0.007273, -1.296573, -2.621487, -0.794329, 1.570796, 1.578069],accel_mss,speed_ms,0,blend_radius_m)
    |   movel([0.006993, -1.293765, -2.623147, -0.795477, 1.570796, 1.577789],accel_mss,speed_ms,0,blend_radius_m)
    |   movel([0.007404, -1.290663, -2.624969, -0.796757, 1.570796, 1.578200],accel_mss,speed_ms,0,blend_radius_m)
    |   movel([0.008595, -1.287303, -2.626929, -0.798157, 1.570796, 1.579391],accel_mss,speed_ms,0,blend_radius_m)
    |   movel([0.010660, -1.283721, -2.629002, -0.799665, 1.570796, 1.581456],accel_mss,speed_ms,0,blend_radius_m)
    |   movel([0.013688, -1.279953, -2.631166, -0.801269, 1.570796, 1.584484],accel_mss,speed_ms,0,blend_radius_m)
    |   movel([0.016195, -1.277394, -2.632626, -0.802369, 1.570796, 1.586991],accel_mss,speed_ms,0,blend_radius_m)
    |   movel([0.018848, -1.275002, -2.633983, -0.803405, 1.570796, 1.589644],accel_mss,speed_ms,0,blend_radius_m)
    |   movel([0.021614, -1.272788, -2.635232, -0.804369, 1.570796, 1.592411],accel_mss,speed_ms,0,blend_radius_m)
    |   movel([0.024476, -1.270775, -2.636363, -0.805251, 1.570796, 1.595272],accel_mss,speed_ms,0,blend_radius_m)
    |   movel([0.027400, -1.268976, -2.637369, -0.806044, 1.570796, 1.598196],accel_mss,speed_ms,0,blend_radius_m)
    |   movel([0.030363, -1.267409, -2.638242, -0.806737, 1.570796, 1.601159],accel_mss,speed_ms,0,blend_radius_m)
    |   movel([0.033337, -1.266091, -2.638975, -0.807323, 1.570796, 1.604133],accel_mss,speed_ms,0,blend_radius_m)
    |   movel([0.036293, -1.265035, -2.639560, -0.807794, 1.570796, 1.607090],accel_mss,speed_ms,0,blend_radius_m)
    |   movel([0.039204, -1.264261, -2.639988, -0.808140, 1.570796, 1.610000],accel_mss,speed_ms,0,blend_radius_m)
    |   movel([0.042042, -1.263780, -2.640253, -0.808356, 1.570796, 1.612839],accel_mss,speed_ms,0,blend_radius_m)
    |   movel([0.044780, -1.263611, -2.640347, -0.808432, 1.570796, 1.615576],accel_mss,speed_ms,0,blend_radius_m)
    |   movel([0.047390, -1.263765, -2.640262, -0.808362, 1.570796, 1.618187],accel_mss,speed_ms,0,blend_radius_m)
    |   movel([0.049843, -1.264256, -2.639991, -0.808142, 1.570796, 1.620640],accel_mss,speed_ms,0,blend_radius_m)
    |   movel([0.052116, -1.265094, -2.639527, -0.807768, 1.570796, 1.622912],accel_mss,speed_ms,0,blend_radius_m)
    |   movel([0.054178, -1.266295, -2.638862, -0.807233, 1.570796, 1.624974],accel_mss,speed_ms,0,blend_radius_m)
    |   movel([0.056005, -1.267868, -2.637987, -0.806534, 1.570796, 1.626801],accel_mss,speed_ms,0,blend_radius_m)
    |   movel([0.057181, -1.269999, -2.636797, -0.805593, 1.570796, 1.627977],accel_mss,speed_ms,0,blend_radius_m)
    |   movel([0.057879, -1.272726, -2.635267, -0.804396, 1.570796, 1.628675],accel_mss,speed_ms,0,blend_radius_m)
    |   movel([0.058316, -1.275175, -2.633885, -0.803329, 1.570796, 1.629113],accel_mss,speed_ms,0,blend_radius_m)
    |   movel([0.058712, -1.276482, -2.633144, -0.802763, 1.570796, 1.629508],accel_mss,speed_ms,0,blend_radius_m)
    |   movel([0.059911, -1.276686, -2.633028, -0.802675, 1.570796, 1.630707],accel_mss,speed_ms,0,blend_radius_m)
    |   movel([0.062107, -1.276584, -2.633086, -0.802719, 1.570796, 1.632904],accel_mss,speed_ms,0,blend_radius_m)
    |   movel([0.064531, -1.276472, -2.633149, -0.802767, 1.570796, 1.635328],accel_mss,speed_ms,0,blend_radius_m)
    |   movel([0.066410, -1.276639, -2.633055, -0.802695, 1.570796, 1.637207],accel_mss,speed_ms,0,blend_radius_m)
    |   movel([0.068473, -1.277486, -2.632573, -0.802330, 1.570796, 1.639269],accel_mss,speed_ms,0,blend_radius_m)
    |   movel([0.070102, -1.278648, -2.631911, -0.801829, 1.570796, 1.640898],accel_mss,speed_ms,0,blend_radius_m)
    |   movel([0.071312, -1.280091, -2.631088, -0.801211, 1.570796, 1.642108],accel_mss,speed_ms,0,blend_radius_m)
    |   movel([0.072122, -1.281773, -2.630124, -0.800493, 1.570796, 1.642918],accel_mss,speed_ms,0,blend_radius_m)
    |   movel([0.072552, -1.283657, -2.629039, -0.799693, 1.570796, 1.643348],accel_mss,speed_ms,0,blend_radius_m)
    |   movel([0.072619, -1.285703, -2.627857, -0.798829, 1.570796, 1.643415],accel_mss,speed_ms,0,blend_radius_m)
    |   movel([0.072345, -1.287875, -2.626596, -0.797918, 1.570796, 1.643141],accel_mss,speed_ms,0,blend_radius_m)
    |   movel([0.071746, -1.290135, -2.625278, -0.796976, 1.570796, 1.642542],accel_mss,speed_ms,0,blend_radius_m)
    |   movel([0.070840, -1.292450, -2.623921, -0.796018, 1.570796, 1.641636],accel_mss,speed_ms,0,blend_radius_m)
    |   movel([0.069646, -1.294782, -2.622547, -0.795060, 1.570796, 1.640443],accel_mss,speed_ms,0,blend_radius_m)
    |   movel([0.068183, -1.297097, -2.621176, -0.794116, 1.570796, 1.638979],accel_mss,speed_ms,0,blend_radius_m)
    |   speed_ms = 0.003
    |   movel([0.068183, -1.290226, -2.617885, -0.804278, 1.570796, 1.638979],accel_mss,speed_ms,0,blend_radius_m)
    |   speed_ms = 0.05
    |   movel([0.068183, -1.263928, -2.604442, -0.844019, 1.570796, 1.638979],accel_mss,speed_ms,0,blend_radius_m)
    |   #M_RunCode9
    |   movel([0.084832, -1.255809, -2.609002, -0.847577, 1.570796, 1.655628],accel_mss,speed_ms,0,blend_radius_m)
    |   #M_RunCode3
    |   movel([0.084832, -1.282218, -2.622552, -0.807619, 1.570796, 1.655628],accel_mss,speed_ms,0,blend_radius_m)
    |   speed_ms = 0.003
    |   movel([0.084832, -1.289121, -2.625870, -0.797398, 1.570796, 1.655628],accel_mss,speed_ms,0,blend_radius_m)
    |   speed_ms = 0.02
    |   movel([0.084749, -1.287403, -2.626871, -0.798115, 1.570796, 1.655546],accel_mss,speed_ms,0,blend_radius_m)
    |   movel([0.085169, -1.283656, -2.629040, -0.799693, 1.570796, 1.655966],accel_mss,speed_ms,0,blend_radius_m)
    |   movel([0.085368, -1.280083, -2.631092, -0.801214, 1.570796, 1.656164],accel_mss,speed_ms,0,blend_radius_m)
    |   movel([0.085006, -1.278588, -2.631946, -0.801855, 1.570796, 1.655802],accel_mss,speed_ms,0,blend_radius_m)
    |   movel([0.084130, -1.277409, -2.632617, -0.802363, 1.570796, 1.654926],accel_mss,speed_ms,0,blend_radius_m)
    |   movel([0.085162, -1.277896, -2.632340, -0.802153, 1.570796, 1.655959],accel_mss,speed_ms,0,blend_radius_m)
    |   movel([0.086624, -1.279202, -2.631596, -0.801592, 1.570796, 1.657421],accel_mss,speed_ms,0,blend_radius_m)
    |   movel([0.087426, -1.280846, -2.630655, -0.800888, 1.570796, 1.658223],accel_mss,speed_ms,0,blend_radius_m)
    |   movel([0.087774, -1.282723, -2.629577, -0.800088, 1.570796, 1.658570],accel_mss,speed_ms,0,blend_radius_m)
    |   movel([0.087872, -1.284732, -2.628419, -0.799238, 1.570796, 1.658668],accel_mss,speed_ms,0,blend_radius_m)
    |   movel([0.088130, -1.288736, -2.626095, -0.797558, 1.570796, 1.658927],accel_mss,speed_ms,0,blend_radius_m)
    |   movel([0.088691, -1.290538, -2.625042, -0.796809, 1.570796, 1.659487],accel_mss,speed_ms,0,blend_radius_m)
    |   movel([0.089802, -1.292076, -2.624141, -0.796172, 1.570796, 1.660598],accel_mss,speed_ms,0,blend_radius_m)
    |   movel([0.091542, -1.293396, -2.623364, -0.795629, 1.570796, 1.662339],accel_mss,speed_ms,0,blend_radius_m)
    |   movel([0.092585, -1.293988, -2.623015, -0.795385, 1.570796, 1.663382],accel_mss,speed_ms,0,blend_radius_m)
    |   movel([0.093338, -1.294158, -2.622915, -0.795316, 1.570796, 1.664134],accel_mss,speed_ms,0,blend_radius_m)
    |   movel([0.094586, -1.293197, -2.623481, -0.795710, 1.570796, 1.665383],accel_mss,speed_ms,0,blend_radius_m)
    |   movel([0.095633, -1.292448, -2.623922, -0.796019, 1.570796, 1.666429],accel_mss,speed_ms,0,blend_radius_m)
    |   movel([0.096777, -1.291840, -2.624279, -0.796270, 1.570796, 1.667573],accel_mss,speed_ms,0,blend_radius_m)
    |   movel([0.099080, -1.291066, -2.624733, -0.796590, 1.570796, 1.669877],accel_mss,speed_ms,0,blend_radius_m)
    |   movel([0.100789, -1.290798, -2.624890, -0.796701, 1.570796, 1.671585],accel_mss,speed_ms,0,blend_radius_m)
    |   movel([0.102040, -1.290940, -2.624807, -0.796642, 1.570796, 1.672836],accel_mss,speed_ms,0,blend_radius_m)
    |   movel([0.102975, -1.291401, -2.624537, -0.796451, 1.570796, 1.673772],accel_mss,speed_ms,0,blend_radius_m)
    |   movel([0.104468, -1.292911, -2.623649, -0.795828, 1.570796, 1.675264],accel_mss,speed_ms,0,blend_radius_m)
    |   movel([0.106404, -1.294598, -2.622655, -0.795135, 1.570796, 1.677201],accel_mss,speed_ms,0,blend_radius_m)
    |   movel([0.109606, -1.296266, -2.621669, -0.794454, 1.570796, 1.680403],accel_mss,speed_ms,0,blend_radius_m)
    |   movel([0.112907, -1.297793, -2.620762, -0.793833, 1.570796, 1.683704],accel_mss,speed_ms,0,blend_radius_m)
    |   movel([0.116032, -1.299510, -2.619740, -0.793140, 1.570796, 1.686828],accel_mss,speed_ms,0,blend_radius_m)
    |   movel([0.118709, -1.301726, -2.618414, -0.792249, 1.570796, 1.689506],accel_mss,speed_ms,0,blend_radius_m)
    |   movel([0.119830, -1.303225, -2.617513, -0.791650, 1.570796, 1.690626],accel_mss,speed_ms,0,blend_radius_m)
    |   movel([0.120691, -1.304911, -2.616498, -0.790980, 1.570796, 1.691487],accel_mss,speed_ms,0,blend_radius_m)
    |   movel([0.121877, -1.308632, -2.614242, -0.789515, 1.570796, 1.692674],accel_mss,speed_ms,0,blend_radius_m)
    |   movel([0.122757, -1.312481, -2.611890, -0.788018, 1.570796, 1.693553],accel_mss,speed_ms,0,blend_radius_m)
    |   movel([0.123811, -1.316053, -2.609689, -0.786647, 1.570796, 1.694607],accel_mss,speed_ms,0,blend_radius_m)
    |   movel([0.126430, -1.321390, -2.606370, -0.784629, 1.570796, 1.697226],accel_mss,speed_ms,0,blend_radius_m)
    |   movel([0.127627, -1.323620, -2.604972, -0.783797, 1.570796, 1.698423],accel_mss,speed_ms,0,blend_radius_m)
    |   movel([0.128553, -1.325853, -2.603565, -0.782970, 1.570796, 1.699350],accel_mss,speed_ms,0,blend_radius_m)
    |   movel([0.129078, -1.328302, -2.602015, -0.782071, 1.570796, 1.699874],accel_mss,speed_ms,0,blend_radius_m)
    |   movel([0.129056, -1.331181, -2.600182, -0.781025, 1.570796, 1.699852],accel_mss,speed_ms,0,blend_radius_m)
    |   movel([0.128350, -1.334700, -2.597927, -0.779762, 1.570796, 1.699146],accel_mss,speed_ms,0,blend_radius_m)
    |   movel([0.126832, -1.339058, -2.595111, -0.778220, 1.570796, 1.697628],accel_mss,speed_ms,0,blend_radius_m)
    |   movel([0.125204, -1.342608, -2.592798, -0.776983, 1.570796, 1.696001],accel_mss,speed_ms,0,blend_radius_m)
    |   movel([0.123356, -1.345835, -2.590680, -0.775874, 1.570796, 1.694152],accel_mss,speed_ms,0,blend_radius_m)
    |   movel([0.121304, -1.348754, -2.588752, -0.774883, 1.570796, 1.692101],accel_mss,speed_ms,0,blend_radius_m)
    |   movel([0.119062, -1.351387, -2.587003, -0.773999, 1.570796, 1.689858],accel_mss,speed_ms,0,blend_radius_m)
    |   movel([0.116654, -1.353746, -2.585428, -0.773215, 1.570796, 1.687451],accel_mss,speed_ms,0,blend_radius_m)
    |   movel([0.114093, -1.355849, -2.584017, -0.772523, 1.570796, 1.684889],accel_mss,speed_ms,0,blend_radius_m)
    |   movel([0.111397, -1.357710, -2.582763, -0.771916, 1.570796, 1.682193],accel_mss,speed_ms,0,blend_radius_m)
    |   movel([0.108579, -1.359344, -2.581658, -0.771387, 1.570796, 1.679376],accel_mss,speed_ms,0,blend_radius_m)
    |   movel([0.105663, -1.360764, -2.580696, -0.770930, 1.570796, 1.676459],accel_mss,speed_ms,0,blend_radius_m)
    |   movel([0.102658, -1.361987, -2.579864, -0.770538, 1.570796, 1.673454],accel_mss,speed_ms,0,blend_radius_m)
    |   movel([0.096454, -1.363889, -2.578566, -0.769934, 1.570796, 1.667250],accel_mss,speed_ms,0,blend_radius_m)
    |   movel([0.090104, -1.365152, -2.577702, -0.769535, 1.570796, 1.660901],accel_mss,speed_ms,0,blend_radius_m)
    |   movel([0.083742, -1.365874, -2.577206, -0.769308, 1.570796, 1.654539],accel_mss,speed_ms,0,blend_radius_m)
    |   movel([0.077904, -1.366063, -2.577077, -0.769249, 1.570796, 1.648700],accel_mss,speed_ms,0,blend_radius_m)
    |   movel([0.070465, -1.366204, -2.576980, -0.769205, 1.570796, 1.641261],accel_mss,speed_ms,0,blend_radius_m)
    |   movel([0.062092, -1.366757, -2.576600, -0.769032, 1.570796, 1.632888],accel_mss,speed_ms,0,blend_radius_m)
    |   movel([0.057771, -1.367320, -2.576212, -0.768856, 1.570796, 1.628567],accel_mss,speed_ms,0,blend_radius_m)
    |   movel([0.053474, -1.368145, -2.575644, -0.768600, 1.570796, 1.624271],accel_mss,speed_ms,0,blend_radius_m)
    |   movel([0.049300, -1.369279, -2.574861, -0.768249, 1.570796, 1.620097],accel_mss,speed_ms,0,blend_radius_m)
    |   movel([0.045333, -1.370767, -2.573832, -0.767791, 1.570796, 1.616130],accel_mss,speed_ms,0,blend_radius_m)
    |   movel([0.041667, -1.372655, -2.572520, -0.767214, 1.570796, 1.612463],accel_mss,speed_ms,0,blend_radius_m)
    |   movel([0.038396, -1.374981, -2.570897, -0.766511, 1.570796, 1.609192],accel_mss,speed_ms,0,blend_radius_m)
    |   movel([0.036934, -1.376324, -2.569957, -0.766108, 1.570796, 1.607730],accel_mss,speed_ms,0,blend_radius_m)
    |   movel([0.035606, -1.377792, -2.568927, -0.765671, 1.570796, 1.606402],accel_mss,speed_ms,0,blend_radius_m)
    |   movel([0.034420, -1.379388, -2.567802, -0.765199, 1.570796, 1.605216],accel_mss,speed_ms,0,blend_radius_m)
    |   movel([0.033388, -1.381119, -2.566579, -0.764691, 1.570796, 1.604184],accel_mss,speed_ms,0,blend_radius_m)
    |   movel([0.032521, -1.382991, -2.565251, -0.764147, 1.570796, 1.603317],accel_mss,speed_ms,0,blend_radius_m)
    |   movel([0.031827, -1.385007, -2.563815, -0.763567, 1.570796, 1.602623],accel_mss,speed_ms,0,blend_radius_m)
